LIN {X 0,Y 467.875,Z 296.784,A -85,B 0,C 180,E1 -7639.396,E2 -7639.396} C_VEL
LIN {X 0,Y 467.446,Z 305.686,A -85,B 0,C 180,E1 -7640.699,E2 -7640.699} C_VEL
LIN {X 0,Y 467.093,Z 312.847,A -85,B 0,C 180,E1 -7642,E2 -7642} C_VEL
LIN {X 0,Y 466.87,Z 319.224,A -85,B 0,C 180,E1 -7643.479,E2 -7643.479} C_VEL
LIN {X 0,Y 466.784,Z 323.676,A -85,B 0,C 180,E1 -7644.817,E2 -7644.817} C_VEL
LIN {X 0,Y 466.663,Z 325.957,A -85,B 0,C 180,E1 -7645.681,E2 -7645.681} C_VEL
LIN {X 0,Y 466.695,Z 327.806,A -85,B 0,C 180,E1 -7646.546,E2 -7646.546} C_VEL
LIN {X 0,Y 466.646,Z 329.192,A -85,B 0,C 180,E1 -7647.41,E2 -7647.41} C_VEL
LIN {X 0,Y 466.589,Z 330.785,A -85,B 0,C 180,E1 -7649.137,E2 -7649.137} C_VEL
LIN {X 0,Y 466.57,Z 331,A -85,B 0,C 180,E1 -7650,E2 -7650} C_VEL
LIN {X 0,Y 466.589,Z 330.786,A -85,B 0,C 180,E1 -7650.863,E2 -7650.863} C_VEL
LIN {X 0,Y 466.646,Z 329.196,A -85,B 0,C 180,E1 -7652.589,E2 -7652.589} C_VEL
LIN {X 0,Y 466.695,Z 327.81,A -85,B 0,C 180,E1 -7653.453,E2 -7653.453} C_VEL
LIN {X 0,Y 466.703,Z 324.896,A -85,B 0,C 180,E1 -7654.751,E2 -7654.751} C_VEL
LIN {X 0,Y 466.84,Z 320.949,A -85,B 0,C 180,E1 -7656.049,E2 -7656.049} C_VEL
LIN {X 0,Y 466.998,Z 314.876,A -85,B 0,C 180,E1 -7657.567,E2 -7657.567} C_VEL
LIN {X 0,Y 467.35,Z 308.236,A -85,B 0,C 180,E1 -7658.867,E2 -7658.867} C_VEL
LIN {X 0,Y 467.737,Z 299.994,A -85,B 0,C 180,E1 -7660.169,E2 -7660.169} C_VEL
LIN {X 0,Y 468.123,Z 291.523,A -85,B 0,C 180,E1 -7661.254,E2 -7661.254} C_VEL
LIN {X 0,Y 468.66,Z 281.242,A -85,B 0,C 180,E1 -7662.319,E2 -7662.319} C_VEL
LIN {X 0,Y 469.099,Z 269.657,A -85,B 0,C 180,E1 -7663.284,E2 -7663.284} C_VEL
LIN {X 0,Y 469.623,Z 257.36,A -85,B 0,C 180,E1 -7664.074,E2 -7664.074} C_VEL
LIN {X 0,Y 470.109,Z 245.016,A -85,B 0,C 180,E1 -7664.667,E2 -7664.667} C_VEL
LIN {X 0,Y 469.597,Z 238.804,A -85,B 0,C 180,E1 -7664.922,E2 -7664.922} C_VEL
LIN {X 0,Y 467.324,Z 225.956,A -85,B 0,C 180,E1 -7665.358,E2 -7665.358} C_VEL
LIN {X 0,Y 467.08,Z 224.269,A -85,B 0,C 180,E1 -7665.42,E2 -7665.42} C_VEL
LIN {X 0,Y 467.234,Z 216.192,A -85,B 0,C 180,E1 -7668.625,E2 -7668.625} C_VEL
LIN {X 0,Y 467.417,Z 208.755,A -85,B 0,C 180,E1 -7671.615,E2 -7671.615} C_VEL
LIN {X 0,Y 467.625,Z 201.974,A -85,B 0,C 180,E1 -7674.412,E2 -7674.412} C_VEL
LIN {X 0,Y 467.942,Z 194.095,A -85,B 0,C 180,E1 -7677.748,E2 -7677.748} C_VEL
LIN {X 0,Y 468.191,Z 187.326,A -85,B 0,C 180,E1 -7680.688,E2 -7680.688} C_VEL
LIN {X 0,Y 468.489,Z 180.565,A -85,B 0,C 180,E1 -7683.714,E2 -7683.714} C_VEL
LIN {X 0,Y 468.556,Z 175.849,A -85,B 0,C 180,E1 -7685.908,E2 -7685.908} C_VEL
LIN {X 0,Y 467.806,Z 170.377,A -85,B 0,C 180,E1 -7688.628,E2 -7688.628} C_VEL
LIN {X 0,Y 467.581,Z 169.245,A -85,B 0,C 180,E1 -7689.283,E2 -7689.283} C_VEL
LIN {X 0,Y 467.586,Z 169.242,A -85,B 0,C 180,E1 -7692.567,E2 -7692.567} C_VEL
LIN {X 0,Y 467.565,Z 169.245,A -85,B 0,C 180,E1 -7695.052,E2 -7695.052} C_VEL
LIN {X 0,Y 467.588,Z 169.24,A -85,B 0,C 180,E1 -7697.44,E2 -7697.44} C_VEL
LIN {X 0,Y 467.549,Z 169.245,A -85,B 0,C 180,E1 -7700.852,E2 -7700.852} C_VEL
LIN {X 0,Y 467.55,Z 169.247,A -85,B 0,C 180,E1 -7704.262,E2 -7704.262} C_VEL
LIN {X 0,Y 467.579,Z 169.241,A -85,B 0,C 180,E1 -7707.321,E2 -7707.321} C_VEL
LIN {X 0,Y 467.569,Z 169.244,A -85,B 0,C 180,E1 -7710.667,E2 -7710.667} C_VEL
LIN {X 0,Y 467.611,Z 169.237,A -85,B 0,C 180,E1 -7713.199,E2 -7713.199} C_VEL
LIN {X 0,Y 467.588,Z 169.238,A -85,B 0,C 180,E1 -7716.469,E2 -7716.469} C_VEL
LIN {X 0,Y 467.62,Z 169.237,A -85,B 0,C 180,E1 -7719.777,E2 -7719.777} C_VEL
LIN {X 0,Y 467.605,Z 169.238,A -85,B 0,C 180,E1 -7722.507,E2 -7722.507} C_VEL
LIN {X 0,Y 467.604,Z 169.239,A -85,B 0,C 180,E1 -7725.196,E2 -7725.196} C_VEL
LIN {X 0,Y 467.653,Z 169.234,A -85,B 0,C 180,E1 -7727.854,E2 -7727.854} C_VEL
LIN {X 0,Y 467.654,Z 169.235,A -85,B 0,C 180,E1 -7731.357,E2 -7731.357} C_VEL
LIN {X 0,Y 467.708,Z 169.223,A -85,B 0,C 180,E1 -7733.962,E2 -7733.962} C_VEL
LIN {X 0,Y 467.856,Z 169.206,A -85,B 0,C 180,E1 -7737.417,E2 -7737.417} C_VEL
LIN {X 0,Y 467.881,Z 169.204,A -85,B 0,C 180,E1 -7740,E2 -7740} C_VEL
LIN {X 0,Y 467.855,Z 169.207,A -85,B 0,C 180,E1 -7742.583,E2 -7742.583} C_VEL
LIN {X 0,Y 467.707,Z 169.224,A -85,B 0,C 180,E1 -7746.038,E2 -7746.038} C_VEL
LIN {X 0,Y 467.654,Z 169.234,A -85,B 0,C 180,E1 -7748.643,E2 -7748.643} C_VEL
LIN {X 0,Y 467.654,Z 169.236,A -85,B 0,C 180,E1 -7752.146,E2 -7752.146} C_VEL
LIN {X 0,Y 467.637,Z 169.236,A -85,B 0,C 180,E1 -7755.695,E2 -7755.695} C_VEL
LIN {X 0,Y 467.615,Z 169.237,A -85,B 0,C 180,E1 -7758.765,E2 -7758.765} C_VEL
LIN {X 0,Y 467.578,Z 169.241,A -85,B 0,C 180,E1 -7761.268,E2 -7761.268} C_VEL
LIN {X 0,Y 467.561,Z 169.247,A -85,B 0,C 180,E1 -7763.944,E2 -7763.944} C_VEL
LIN {X 0,Y 467.611,Z 169.235,A -85,B 0,C 180,E1 -7766.801,E2 -7766.801} C_VEL
LIN {X 0,Y 467.553,Z 169.245,A -85,B 0,C 180,E1 -7769.738,E2 -7769.738} C_VEL
LIN {X 0,Y 467.58,Z 169.242,A -85,B 0,C 180,E1 -7772.759,E2 -7772.759} C_VEL
LIN {X 0,Y 467.543,Z 169.247,A -85,B 0,C 180,E1 -7775.891,E2 -7775.891} C_VEL
LIN {X 0,Y 467.55,Z 169.247,A -85,B 0,C 180,E1 -7779.148,E2 -7779.148} C_VEL
LIN {X 0,Y 467.588,Z 169.24,A -85,B 0,C 180,E1 -7782.56,E2 -7782.56} C_VEL
LIN {X 0,Y 467.57,Z 169.243,A -85,B 0,C 180,E1 -7785.054,E2 -7785.054} C_VEL
LIN {X 0,Y 467.589,Z 169.241,A -85,B 0,C 180,E1 -7787.44,E2 -7787.44} C_VEL
LIN {X 0,Y 467.556,Z 169.245,A -85,B 0,C 180,E1 -7790.853,E2 -7790.853} C_VEL
LIN {X 0,Y 467.512,Z 169.254,A -85,B 0,C 180,E1 -7793.037,E2 -7793.037} C_VEL
LIN {X 0,Y 467.45,Z 169.259,A -85,B 0,C 180,E1 -7794.28,E2 -7794.28} C_VEL
LIN {X 0,Y 467.423,Z 171.585,A -85,B 0,C 180,E1 -7796.199,E2 -7796.199} C_VEL
LIN {X 0,Y 467.378,Z 175.811,A -85,B 0,C 180,E1 -7799.253,E2 -7799.253} C_VEL
LIN {X 0,Y 467.229,Z 180.015,A -85,B 0,C 180,E1 -7802.206,E2 -7802.206} C_VEL
LIN {X 0,Y 467.14,Z 184.191,A -85,B 0,C 180,E1 -7805.087,E2 -7805.087} C_VEL
LIN {X 0,Y 467.047,Z 188.346,A -85,B 0,C 180,E1 -7807.902,E2 -7807.902} C_VEL
LIN {X 0,Y 466.911,Z 192.566,A -85,B 0,C 180,E1 -7810.662,E2 -7810.662} C_VEL
LIN {X 0,Y 466.814,Z 197.398,A -85,B 0,C 180,E1 -7813.714,E2 -7813.714} C_VEL
LIN {X 0,Y 466.697,Z 198.811,A -85,B 0,C 180,E1 -7814.092,E2 -7814.092} C_VEL
LIN {X 0,Y 466.299,Z 202.019,A -85,B 0,C 180,E1 -7814.468,E2 -7814.468} C_VEL
LIN {X 0,Y 465.498,Z 207.579,A -85,B 0,C 180,E1 -7814.817,E2 -7814.817} C_VEL
LIN {X 0,Y 463.951,Z 218.12,A -85,B 0,C 180,E1 -7815.189,E2 -7815.189} C_VEL
LIN {X 0,Y 463.13,Z 225.353,A -85,B 0,C 180,E1 -7815.502,E2 -7815.502} C_VEL
LIN {X 0,Y 462.607,Z 236.688,A -85,B 0,C 180,E1 -7816.157,E2 -7816.157} C_VEL
LIN {X 0,Y 462.159,Z 248.349,A -85,B 0,C 180,E1 -7817.038,E2 -7817.038} C_VEL
LIN {X 0,Y 461.634,Z 258.814,A -85,B 0,C 180,E1 -7818.029,E2 -7818.029} C_VEL
LIN {X 0,Y 461.194,Z 267.362,A -85,B 0,C 180,E1 -7819.019,E2 -7819.019} C_VEL
LIN {X 0,Y 460.79,Z 275.235,A -85,B 0,C 180,E1 -7820.12,E2 -7820.12} C_VEL
LIN {X 0,Y 460.344,Z 282.934,A -85,B 0,C 180,E1 -7821.44,E2 -7821.44} C_VEL
LIN {X 0,Y 460.007,Z 289.993,A -85,B 0,C 180,E1 -7822.98,E2 -7822.98} C_VEL
LIN {X 0,Y 459.888,Z 294.695,A -85,B 0,C 180,E1 -7824.299,E2 -7824.299} C_VEL
LIN {X 0,Y 459.69,Z 298.298,A -85,B 0,C 180,E1 -7825.616,E2 -7825.616} C_VEL
LIN {X 0,Y 459.727,Z 300.157,A -85,B 0,C 180,E1 -7826.494,E2 -7826.494} C_VEL
LIN {X 0,Y 459.617,Z 301.562,A -85,B 0,C 180,E1 -7827.371,E2 -7827.371} C_VEL
LIN {X 0,Y 459.525,Z 303.175,A -85,B 0,C 180,E1 -7829.124,E2 -7829.124} C_VEL
LIN {X 0,Y 459.532,Z 303.41,A -85,B 0,C 180,E1 -7830,E2 -7830} C_VEL
LIN {X 0,Y 459.524,Z 303.224,A -85,B 0,C 180,E1 -7830.877,E2 -7830.877} C_VEL
LIN {X 0,Y 459.617,Z 301.675,A -85,B 0,C 180,E1 -7832.629,E2 -7832.629} C_VEL
LIN {X 0,Y 459.726,Z 300.319,A -85,B 0,C 180,E1 -7833.506,E2 -7833.506} C_VEL
LIN {X 0,Y 459.678,Z 297.461,A -85,B 0,C 180,E1 -7834.824,E2 -7834.824} C_VEL
LIN {X 0,Y 459.946,Z 293.575,A -85,B 0,C 180,E1 -7836.14,E2 -7836.14} C_VEL
LIN {X 0,Y 460.053,Z 288.569,A -85,B 0,C 180,E1 -7837.461,E2 -7837.461} C_VEL
LIN {X 0,Y 460.392,Z 282.263,A -85,B 0,C 180,E1 -7838.781,E2 -7838.781} C_VEL
LIN {X 0,Y 460.813,Z 274.368,A -85,B 0,C 180,E1 -7840.102,E2 -7840.102} C_VEL
LIN {X 0,Y 461.215,Z 266.319,A -85,B 0,C 180,E1 -7841.203,E2 -7841.203} C_VEL
LIN {X 0,Y 461.777,Z 256.494,A -85,B 0,C 180,E1 -7842.303,E2 -7842.303} C_VEL
LIN {X 0,Y 462.242,Z 245.72,A -85,B 0,C 180,E1 -7843.274,E2 -7843.274} C_VEL
LIN {X 0,Y 462.781,Z 234.616,A -85,B 0,C 180,E1 -7844.063,E2 -7844.063} C_VEL
LIN {X 0,Y 463.246,Z 222.652,A -85,B 0,C 180,E1 -7844.721,E2 -7844.721} C_VEL
LIN {X 0,Y 463.261,Z 216.269,A -85,B 0,C 180,E1 -7845.008,E2 -7845.008} C_VEL
LIN {X 0,Y 460.768,Z 203.666,A -85,B 0,C 180,E1 -7845.517,E2 -7845.517} C_VEL
LIN {X 0,Y 459.757,Z 199.146,A -85,B 0,C 180,E1 -7845.666,E2 -7845.666} C_VEL
LIN {X 0,Y 459.844,Z 194.325,A -85,B 0,C 180,E1 -7848.721,E2 -7848.721} C_VEL
LIN {X 0,Y 459.918,Z 190.074,A -85,B 0,C 180,E1 -7851.515,E2 -7851.515} C_VEL
LIN {X 0,Y 460.07,Z 185.88,A -85,B 0,C 180,E1 -7854.359,E2 -7854.359} C_VEL
LIN {X 0,Y 460.171,Z 181.159,A -85,B 0,C 180,E1 -7857.648,E2 -7857.648} C_VEL
LIN {X 0,Y 460.291,Z 177.484,A -85,B 0,C 180,E1 -7860.256,E2 -7860.256} C_VEL
LIN {X 0,Y 460.372,Z 173.244,A -85,B 0,C 180,E1 -7863.338,E2 -7863.338} C_VEL
LIN {X 0,Y 460.43,Z 170.397,A -85,B 0,C 180,E1 -7865.453,E2 -7865.453} C_VEL
LIN {X 0,Y 460.48,Z 170.127,A -85,B 0,C 180,E1 -7867.473,E2 -7867.473} C_VEL
LIN {X 0,Y 460.525,Z 170.12,A -85,B 0,C 180,E1 -7870.266,E2 -7870.266} C_VEL
LIN {X 0,Y 460.505,Z 170.124,A -85,B 0,C 180,E1 -7873.375,E2 -7873.375} C_VEL
LIN {X 0,Y 460.5,Z 170.122,A -85,B 0,C 180,E1 -7876.624,E2 -7876.624} C_VEL
LIN {X 0,Y 460.539,Z 170.116,A -85,B 0,C 180,E1 -7879.731,E2 -7879.731} C_VEL
LIN {X 0,Y 460.482,Z 170.128,A -85,B 0,C 180,E1 -7882.527,E2 -7882.527} C_VEL
LIN {X 0,Y 460.535,Z 170.119,A -85,B 0,C 180,E1 -7885.623,E2 -7885.623} C_VEL
LIN {X 0,Y 460.539,Z 170.12,A -85,B 0,C 180,E1 -7888.744,E2 -7888.744} C_VEL
LIN {X 0,Y 460.583,Z 170.114,A -85,B 0,C 180,E1 -7892.254,E2 -7892.254} C_VEL
LIN {X 0,Y 460.541,Z 170.117,A -85,B 0,C 180,E1 -7894.704,E2 -7894.704} C_VEL
LIN {X 0,Y 460.511,Z 170.121,A -85,B 0,C 180,E1 -7897.571,E2 -7897.571} C_VEL
LIN {X 0,Y 460.569,Z 170.115,A -85,B 0,C 180,E1 -7900.384,E2 -7900.384} C_VEL
LIN {X 0,Y 460.601,Z 170.111,A -85,B 0,C 180,E1 -7904.002,E2 -7904.002} C_VEL
LIN {X 0,Y 460.61,Z 170.111,A -85,B 0,C 180,E1 -7907.666,E2 -7907.666} C_VEL
LIN {X 0,Y 460.61,Z 170.109,A -85,B 0,C 180,E1 -7911.223,E2 -7911.223} C_VEL
LIN {X 0,Y 460.674,Z 170.101,A -85,B 0,C 180,E1 -7913.87,E2 -7913.87} C_VEL
LIN {X 0,Y 460.797,Z 170.087,A -85,B 0,C 180,E1 -7917.377,E2 -7917.377} C_VEL
LIN {X 0,Y 460.855,Z 170.079,A -85,B 0,C 180,E1 -7920,E2 -7920} C_VEL
LIN {X 0,Y 460.799,Z 170.086,A -85,B 0,C 180,E1 -7922.622,E2 -7922.622} C_VEL
LIN {X 0,Y 460.676,Z 170.099,A -85,B 0,C 180,E1 -7926.13,E2 -7926.13} C_VEL
LIN {X 0,Y 460.609,Z 170.113,A -85,B 0,C 180,E1 -7928.777,E2 -7928.777} C_VEL
LIN {X 0,Y 460.636,Z 170.108,A -85,B 0,C 180,E1 -7932.457,E2 -7932.457} C_VEL
LIN {X 0,Y 460.601,Z 170.112,A -85,B 0,C 180,E1 -7935.998,E2 -7935.998} C_VEL
LIN {X 0,Y 460.569,Z 170.114,A -85,B 0,C 180,E1 -7939.616,E2 -7939.616} C_VEL
LIN {X 0,Y 460.511,Z 170.123,A -85,B 0,C 180,E1 -7942.429,E2 -7942.429} C_VEL
LIN {X 0,Y 460.553,Z 170.119,A -85,B 0,C 180,E1 -7945.798,E2 -7945.798} C_VEL
LIN {X 0,Y 460.553,Z 170.117,A -85,B 0,C 180,E1 -7948.233,E2 -7948.233} C_VEL
LIN {X 0,Y 460.522,Z 170.122,A -85,B 0,C 180,E1 -7951.283,E2 -7951.283} C_VEL
LIN {X 0,Y 460.53,Z 170.119,A -85,B 0,C 180,E1 -7954.505,E2 -7954.505} C_VEL
LIN {X 0,Y 460.483,Z 170.129,A -85,B 0,C 180,E1 -7957.625,E2 -7957.625} C_VEL
LIN {X 0,Y 460.531,Z 170.12,A -85,B 0,C 180,E1 -7961.011,E2 -7961.011} C_VEL
LIN {X 0,Y 460.508,Z 170.124,A -85,B 0,C 180,E1 -7964.169,E2 -7964.169} C_VEL
LIN {X 0,Y 460.514,Z 170.12,A -85,B 0,C 180,E1 -7967.1,E2 -7967.1} C_VEL
LIN {X 0,Y 460.542,Z 170.122,A -85,B 0,C 180,E1 -7970.392,E2 -7970.392} C_VEL
LIN {X 0,Y 460.585,Z 170.311,A -85,B 0,C 180,E1 -7970.649,E2 -7970.649} C_VEL
LIN {X 0,Y 461.488,Z 176.003,A -85,B 0,C 180,E1 -7973.563,E2 -7973.563} C_VEL
LIN {X 0,Y 461.531,Z 180.472,A -85,B 0,C 180,E1 -7975.707,E2 -7975.707} C_VEL
LIN {X 0,Y 461.234,Z 187.215,A -85,B 0,C 180,E1 -7978.797,E2 -7978.797} C_VEL
LIN {X 0,Y 460.951,Z 193.981,A -85,B 0,C 180,E1 -7981.794,E2 -7981.794} C_VEL
LIN {X 0,Y 460.653,Z 200.735,A -85,B 0,C 180,E1 -7984.711,E2 -7984.711} C_VEL
LIN {X 0,Y 460.422,Z 207.527,A -85,B 0,C 180,E1 -7987.567,E2 -7987.567} C_VEL
LIN {X 0,Y 460.202,Z 215.596,A -85,B 0,C 180,E1 -7990.878,E2 -7990.878} C_VEL
LIN {X 0,Y 460.029,Z 224.29,A -85,B 0,C 180,E1 -7994.364,E2 -7994.364} C_VEL
LIN {X 0,Y 462.399,Z 237.666,A -85,B 0,C 180,E1 -7994.806,E2 -7994.806} C_VEL
LIN {X 0,Y 463.229,Z 244.803,A -85,B 0,C 180,E1 -7995.109,E2 -7995.109} C_VEL
LIN {X 0,Y 462.786,Z 257.144,A -85,B 0,C 180,E1 -7995.713,E2 -7995.713} C_VEL
LIN {X 0,Y 462.22,Z 269.005,A -85,B 0,C 180,E1 -7996.48,E2 -7996.48} C_VEL
LIN {X 0,Y 461.765,Z 279.345,A -85,B 0,C 180,E1 -7997.334,E2 -7997.334} C_VEL
LIN {X 0,Y 461.267,Z 289.356,A -85,B 0,C 180,E1 -7998.353,E2 -7998.353} C_VEL
LIN {X 0,Y 460.754,Z 298.208,A -85,B 0,C 180,E1 -7999.453,E2 -7999.453} C_VEL
LIN {X 0,Y 460.346,Z 306.844,A -85,B 0,C 180,E1 -8000.775,E2 -8000.775} C_VEL
LIN {X 0,Y 459.98,Z 313.745,A -85,B 0,C 180,E1 -8002.096,E2 -8002.096} C_VEL
LIN {X 0,Y 459.8,Z 319.492,A -85,B 0,C 180,E1 -8003.475,E2 -8003.475} C_VEL
LIN {X 0,Y 459.701,Z 323.619,A -85,B 0,C 180,E1 -8004.737,E2 -8004.737} C_VEL
LIN {X 0,Y 459.58,Z 325.915,A -85,B 0,C 180,E1 -8005.615,E2 -8005.615} C_VEL
LIN {X 0,Y 459.591,Z 327.779,A -85,B 0,C 180,E1 -8006.493,E2 -8006.493} C_VEL
LIN {X 0,Y 459.57,Z 329.176,A -85,B 0,C 180,E1 -8007.37,E2 -8007.37} C_VEL
LIN {X 0,Y 459.494,Z 330.779,A -85,B 0,C 180,E1 -8009.123,E2 -8009.123} C_VEL
LIN {X 0,Y 459.474,Z 330.994,A -85,B 0,C 180,E1 -8010,E2 -8010} C_VEL
LIN {X 0,Y 459.494,Z 330.779,A -85,B 0,C 180,E1 -8010.876,E2 -8010.876} C_VEL
LIN {X 0,Y 459.57,Z 329.179,A -85,B 0,C 180,E1 -8012.629,E2 -8012.629} C_VEL
LIN {X 0,Y 459.591,Z 327.783,A -85,B 0,C 180,E1 -8013.507,E2 -8013.507} C_VEL
LIN {X 0,Y 459.634,Z 324.846,A -85,B 0,C 180,E1 -8014.824,E2 -8014.824} C_VEL
LIN {X 0,Y 459.758,Z 320.873,A -85,B 0,C 180,E1 -8016.142,E2 -8016.142} C_VEL
LIN {X 0,Y 459.929,Z 314.76,A -85,B 0,C 180,E1 -8017.684,E2 -8017.684} C_VEL
LIN {X 0,Y 460.305,Z 308.084,A -85,B 0,C 180,E1 -8019.003,E2 -8019.003} C_VEL
LIN {X 0,Y 460.698,Z 299.799,A -85,B 0,C 180,E1 -8020.326,E2 -8020.326} C_VEL
LIN {X 0,Y 461.133,Z 291.309,A -85,B 0,C 180,E1 -8021.427,E2 -8021.427} C_VEL
LIN {X 0,Y 461.678,Z 281.197,A -85,B 0,C 180,E1 -8022.493,E2 -8022.493} C_VEL
LIN {X 0,Y 462.116,Z 270.731,A -85,B 0,C 180,E1 -8023.388,E2 -8023.388} C_VEL
LIN {X 0,Y 462.631,Z 259.068,A -85,B 0,C 180,E1 -8024.179,E2 -8024.179} C_VEL
LIN {X 0,Y 463.133,Z 247.407,A -85,B 0,C 180,E1 -8024.781,E2 -8024.781} C_VEL
LIN {X 0,Y 463.006,Z 241.858,A -85,B 0,C 180,E1 -8025.02,E2 -8025.02} C_VEL
LIN {X 0,Y 460.834,Z 229.016,A -85,B 0,C 180,E1 -8025.501,E2 -8025.501} C_VEL
LIN {X 0,Y 460.019,Z 224.117,A -85,B 0,C 180,E1 -8025.662,E2 -8025.662} C_VEL
LIN {X 0,Y 460.2,Z 215.549,A -85,B 0,C 180,E1 -8029.121,E2 -8029.121} C_VEL
LIN {X 0,Y 460.42,Z 207.462,A -85,B 0,C 180,E1 -8032.433,E2 -8032.433} C_VEL
LIN {X 0,Y 460.738,Z 199.434,A -85,B 0,C 180,E1 -8035.845,E2 -8035.845} C_VEL
LIN {X 0,Y 460.986,Z 192.849,A -85,B 0,C 180,E1 -8038.7,E2 -8038.7} C_VEL
LIN {X 0,Y 461.258,Z 186.702,A -85,B 0,C 180,E1 -8041.433,E2 -8041.433} C_VEL
LIN {X 0,Y 461.584,Z 179.604,A -85,B 0,C 180,E1 -8044.695,E2 -8044.695} C_VEL
LIN {X 0,Y 461.493,Z 175.986,A -85,B 0,C 180,E1 -8046.436,E2 -8046.436} C_VEL
LIN {X 0,Y 460.549,Z 170.122,A -85,B 0,C 180,E1 -8049.481,E2 -8049.481} C_VEL
LIN {X 0,Y 460.522,Z 170.123,A -85,B 0,C 180,E1 -8052.181,E2 -8052.181} C_VEL
LIN {X 0,Y 460.512,Z 170.122,A -85,B 0,C 180,E1 -8055.411,E2 -8055.411} C_VEL
LIN {X 0,Y 460.531,Z 170.12,A -85,B 0,C 180,E1 -8058.397,E2 -8058.397} C_VEL
LIN {X 0,Y 460.503,Z 170.12,A -85,B 0,C 180,E1 -8061.264,E2 -8061.264} C_VEL
LIN {X 0,Y 460.502,Z 170.123,A -85,B 0,C 180,E1 -8064.554,E2 -8064.554} C_VEL
LIN {X 0,Y 460.529,Z 170.121,A -85,B 0,C 180,E1 -8067.715,E2 -8067.715} C_VEL
LIN {X 0,Y 460.538,Z 170.119,A -85,B 0,C 180,E1 -8070.769,E2 -8070.769} C_VEL
LIN {X 0,Y 460.554,Z 170.117,A -85,B 0,C 180,E1 -8073.734,E2 -8073.734} C_VEL
LIN {X 0,Y 460.542,Z 170.115,A -85,B 0,C 180,E1 -8076.624,E2 -8076.624} C_VEL
LIN {X 0,Y 460.549,Z 170.119,A -85,B 0,C 180,E1 -8079.453,E2 -8079.453} C_VEL
LIN {X 0,Y 460.556,Z 170.117,A -85,B 0,C 180,E1 -8082.23,E2 -8082.23} C_VEL
LIN {X 0,Y 460.563,Z 170.117,A -85,B 0,C 180,E1 -8084.965,E2 -8084.965} C_VEL
LIN {X 0,Y 460.606,Z 170.11,A -85,B 0,C 180,E1 -8088.559,E2 -8088.559} C_VEL
LIN {X 0,Y 460.606,Z 170.112,A -85,B 0,C 180,E1 -8091.223,E2 -8091.223} C_VEL
LIN {X 0,Y 460.672,Z 170.099,A -85,B 0,C 180,E1 -8093.87,E2 -8093.87} C_VEL
LIN {X 0,Y 460.796,Z 170.086,A -85,B 0,C 180,E1 -8097.378,E2 -8097.378} C_VEL
LIN {X 0,Y 460.852,Z 170.079,A -85,B 0,C 180,E1 -8100,E2 -8100} C_VEL
LIN {X 0,Y 460.796,Z 170.087,A -85,B 0,C 180,E1 -8102.623,E2 -8102.623} C_VEL
LIN {X 0,Y 460.672,Z 170.101,A -85,B 0,C 180,E1 -8106.13,E2 -8106.13} C_VEL
LIN {X 0,Y 460.606,Z 170.11,A -85,B 0,C 180,E1 -8108.777,E2 -8108.777} C_VEL
LIN {X 0,Y 460.611,Z 170.11,A -85,B 0,C 180,E1 -8112.445,E2 -8112.445} C_VEL
LIN {X 0,Y 460.598,Z 170.112,A -85,B 0,C 180,E1 -8115.998,E2 -8115.998} C_VEL
LIN {X 0,Y 460.569,Z 170.114,A -85,B 0,C 180,E1 -8118.902,E2 -8118.902} C_VEL
LIN {X 0,Y 460.514,Z 170.121,A -85,B 0,C 180,E1 -8121.486,E2 -8121.486} C_VEL
LIN {X 0,Y 460.529,Z 170.118,A -85,B 0,C 180,E1 -8124.333,E2 -8124.333} C_VEL
LIN {X 0,Y 460.587,Z 170.114,A -85,B 0,C 180,E1 -8127.748,E2 -8127.748} C_VEL
LIN {X 0,Y 460.519,Z 170.123,A -85,B 0,C 180,E1 -8131.283,E2 -8131.283} C_VEL
LIN {X 0,Y 460.527,Z 170.12,A -85,B 0,C 180,E1 -8134.505,E2 -8134.505} C_VEL
LIN {X 0,Y 460.482,Z 170.127,A -85,B 0,C 180,E1 -8137.625,E2 -8137.625} C_VEL
LIN {X 0,Y 460.537,Z 170.116,A -85,B 0,C 180,E1 -8140.269,E2 -8140.269} C_VEL
LIN {X 0,Y 460.497,Z 170.123,A -85,B 0,C 180,E1 -8143.376,E2 -8143.376} C_VEL
LIN {X 0,Y 460.5,Z 170.125,A -85,B 0,C 180,E1 -8146.625,E2 -8146.625} C_VEL
LIN {X 0,Y 460.538,Z 170.118,A -85,B 0,C 180,E1 -8149.732,E2 -8149.732} C_VEL
LIN {X 0,Y 460.491,Z 170.125,A -85,B 0,C 180,E1 -8152.526,E2 -8152.526} C_VEL
LIN {X 0,Y 460.371,Z 170.266,A -85,B 0,C 180,E1 -8154.542,E2 -8154.542} C_VEL
LIN {X 0,Y 460.345,Z 173.703,A -85,B 0,C 180,E1 -8157.106,E2 -8157.106} C_VEL
LIN {X 0,Y 460.29,Z 177.344,A -85,B 0,C 180,E1 -8159.744,E2 -8159.744} C_VEL
LIN {X 0,Y 460.169,Z 181.546,A -85,B 0,C 180,E1 -8162.731,E2 -8162.731} C_VEL
LIN {X 0,Y 460.071,Z 185.729,A -85,B 0,C 180,E1 -8165.642,E2 -8165.642} C_VEL
LIN {X 0,Y 459.963,Z 190.324,A -85,B 0,C 180,E1 -8168.757,E2 -8168.757} C_VEL
LIN {X 0,Y 459.794,Z 195.597,A -85,B 0,C 180,E1 -8172.2,E2 -8172.2} C_VEL
LIN {X 0,Y 459.79,Z 199.144,A -85,B 0,C 180,E1 -8174.427,E2 -8174.427} C_VEL
LIN {X 0,Y 462.626,Z 212.526,A -85,B 0,C 180,E1 -8174.921,E2 -8174.921} C_VEL
LIN {X 0,Y 463.362,Z 218.158,A -85,B 0,C 180,E1 -8175.17,E2 -8175.17} C_VEL
LIN {X 0,Y 463.13,Z 225.353,A -85,B 0,C 180,E1 -8175.502,E2 -8175.502} C_VEL
LIN {X 0,Y 462.255,Z 230.79,A -85,B 0,C 180,E1 -8175.768,E2 -8175.768} C_VEL
LIN {X 0,Y 459.168,Z 239.456,A -85,B 0,C 180,E1 -8176.227,E2 -8176.227} C_VEL
LIN {X 0,Y 456.036,Z 247.721,A -85,B 0,C 180,E1 -8176.781,E2 -8176.781} C_VEL
LIN {X 0,Y 455.097,Z 252.526,A -85,B 0,C 180,E1 -8177.194,E2 -8177.194} C_VEL
LIN {X 0,Y 454.553,Z 262.05,A -85,B 0,C 180,E1 -8178.179,E2 -8178.179} C_VEL
LIN {X 0,Y 454.07,Z 270.894,A -85,B 0,C 180,E1 -8179.296,E2 -8179.296} C_VEL
LIN {X 0,Y 453.584,Z 279.522,A -85,B 0,C 180,E1 -8180.637,E2 -8180.637} C_VEL
LIN {X 0,Y 453.133,Z 286.4,A -85,B 0,C 180,E1 -8181.976,E2 -8181.976} C_VEL
LIN {X 0,Y 452.899,Z 291.798,A -85,B 0,C 180,E1 -8183.287,E2 -8183.287} C_VEL
LIN {X 0,Y 452.702,Z 296.226,A -85,B 0,C 180,E1 -8184.656,E2 -8184.656} C_VEL
LIN {X 0,Y 452.599,Z 298.513,A -85,B 0,C 180,E1 -8185.547,E2 -8185.547} C_VEL
LIN {X 0,Y 452.641,Z 300.371,A -85,B 0,C 180,E1 -8186.439,E2 -8186.439} C_VEL
LIN {X 0,Y 452.544,Z 301.775,A -85,B 0,C 180,E1 -8187.33,E2 -8187.33} C_VEL
LIN {X 0,Y 452.432,Z 303.389,A -85,B 0,C 180,E1 -8189.11,E2 -8189.11} C_VEL
LIN {X 0,Y 452.437,Z 303.623,A -85,B 0,C 180,E1 -8190,E2 -8190} C_VEL
LIN {X 0,Y 452.432,Z 303.437,A -85,B 0,C 180,E1 -8190.89,E2 -8190.89} C_VEL
LIN {X 0,Y 452.544,Z 301.887,A -85,B 0,C 180,E1 -8192.671,E2 -8192.671} C_VEL
LIN {X 0,Y 452.64,Z 300.531,A -85,B 0,C 180,E1 -8193.561,E2 -8193.561} C_VEL
LIN {X 0,Y 452.609,Z 297.672,A -85,B 0,C 180,E1 -8194.899,E2 -8194.899} C_VEL
LIN {X 0,Y 452.874,Z 293.787,A -85,B 0,C 180,E1 -8196.237,E2 -8196.237} C_VEL
LIN {X 0,Y 452.998,Z 288.781,A -85,B 0,C 180,E1 -8197.578,E2 -8197.578} C_VEL
LIN {X 0,Y 453.381,Z 282.474,A -85,B 0,C 180,E1 -8198.918,E2 -8198.918} C_VEL
LIN {X 0,Y 453.807,Z 274.578,A -85,B 0,C 180,E1 -8200.259,E2 -8200.259} C_VEL
LIN {X 0,Y 454.253,Z 266.529,A -85,B 0,C 180,E1 -8201.377,E2 -8201.377} C_VEL
LIN {X 0,Y 454.831,Z 256.703,A -85,B 0,C 180,E1 -8202.494,E2 -8202.494} C_VEL
LIN {X 0,Y 455.391,Z 245.359,A -85,B 0,C 180,E1 -8203.523,E2 -8203.523} C_VEL
LIN {X 0,Y 455.901,Z 234.822,A -85,B 0,C 180,E1 -8204.28,E2 -8204.28} C_VEL
LIN {X 0,Y 456.399,Z 222.855,A -85,B 0,C 180,E1 -8204.947,E2 -8204.947} C_VEL
LIN {X 0,Y 456.282,Z 216.534,A -85,B 0,C 180,E1 -8205.24,E2 -8205.24} C_VEL
LIN {X 0,Y 453.764,Z 204.067,A -85,B 0,C 180,E1 -8205.757,E2 -8205.757} C_VEL
LIN {X 0,Y 452.697,Z 199.349,A -85,B 0,C 180,E1 -8205.918,E2 -8205.918} C_VEL
LIN {X 0,Y 452.782,Z 194.512,A -85,B 0,C 180,E1 -8209.024,E2 -8209.024} C_VEL
LIN {X 0,Y 452.884,Z 190.245,A -85,B 0,C 180,E1 -8211.866,E2 -8211.866} C_VEL
LIN {X 0,Y 453.008,Z 186.038,A -85,B 0,C 180,E1 -8214.764,E2 -8214.764} C_VEL
LIN {X 0,Y 453.119,Z 181.66,A -85,B 0,C 180,E1 -8217.86,E2 -8217.86} C_VEL
LIN {X 0,Y 453.26,Z 177.606,A -85,B 0,C 180,E1 -8220.776,E2 -8220.776} C_VEL
LIN {X 0,Y 453.355,Z 173.347,A -85,B 0,C 180,E1 -8223.923,E2 -8223.923} C_VEL
LIN {X 0,Y 453.386,Z 171.926,A -85,B 0,C 180,E1 -8224.998,E2 -8224.998} C_VEL
LIN {X 0,Y 453.405,Z 171.009,A -85,B 0,C 180,E1 -8226.29,E2 -8226.29} C_VEL
LIN {X 0,Y 453.442,Z 171.003,A -85,B 0,C 180,E1 -8229.455,E2 -8229.455} C_VEL
LIN {X 0,Y 453.45,Z 171.002,A -85,B 0,C 180,E1 -8231.931,E2 -8231.931} C_VEL
LIN {X 0,Y 453.486,Z 170.998,A -85,B 0,C 180,E1 -8235.471,E2 -8235.471} C_VEL
LIN {X 0,Y 453.481,Z 170.995,A -85,B 0,C 180,E1 -8238.209,E2 -8238.209} C_VEL
LIN {X 0,Y 453.465,Z 171.003,A -85,B 0,C 180,E1 -8240.798,E2 -8240.798} C_VEL
LIN {X 0,Y 453.444,Z 171.001,A -85,B 0,C 180,E1 -8243.916,E2 -8243.916} C_VEL
LIN {X 0,Y 453.479,Z 170.999,A -85,B 0,C 180,E1 -8247.151,E2 -8247.151} C_VEL
LIN {X 0,Y 453.476,Z 170.998,A -85,B 0,C 180,E1 -8250.268,E2 -8250.268} C_VEL
LIN {X 0,Y 453.503,Z 170.993,A -85,B 0,C 180,E1 -8253.294,E2 -8253.294} C_VEL
LIN {X 0,Y 453.499,Z 170.998,A -85,B 0,C 180,E1 -8256.238,E2 -8256.238} C_VEL
LIN {X 0,Y 453.483,Z 170.996,A -85,B 0,C 180,E1 -8259.118,E2 -8259.118} C_VEL
LIN {X 0,Y 453.505,Z 170.995,A -85,B 0,C 180,E1 -8261.944,E2 -8261.944} C_VEL
LIN {X 0,Y 453.541,Z 170.99,A -85,B 0,C 180,E1 -8264.726,E2 -8264.726} C_VEL
LIN {X 0,Y 453.559,Z 170.987,A -85,B 0,C 180,E1 -8268.379,E2 -8268.379} C_VEL
LIN {X 0,Y 453.577,Z 170.984,A -85,B 0,C 180,E1 -8271.086,E2 -8271.086} C_VEL
LIN {X 0,Y 453.64,Z 170.977,A -85,B 0,C 180,E1 -8273.774,E2 -8273.774} C_VEL
LIN {X 0,Y 453.741,Z 170.966,A -85,B 0,C 180,E1 -8277.337,E2 -8277.337} C_VEL
LIN {X 0,Y 453.825,Z 170.954,A -85,B 0,C 180,E1 -8280,E2 -8280} C_VEL
LIN {X 0,Y 453.743,Z 170.965,A -85,B 0,C 180,E1 -8282.663,E2 -8282.663} C_VEL
LIN {X 0,Y 453.642,Z 170.975,A -85,B 0,C 180,E1 -8286.226,E2 -8286.226} C_VEL
LIN {X 0,Y 453.577,Z 170.987,A -85,B 0,C 180,E1 -8288.914,E2 -8288.914} C_VEL
LIN {X 0,Y 453.603,Z 170.984,A -85,B 0,C 180,E1 -8292.551,E2 -8292.551} C_VEL
LIN {X 0,Y 453.545,Z 170.99,A -85,B 0,C 180,E1 -8296.196,E2 -8296.196} C_VEL
LIN {X 0,Y 453.518,Z 170.992,A -85,B 0,C 180,E1 -8299.039,E2 -8299.039} C_VEL
LIN {X 0,Y 453.477,Z 170.997,A -85,B 0,C 180,E1 -8301.836,E2 -8301.836} C_VEL
LIN {X 0,Y 453.501,Z 170.994,A -85,B 0,C 180,E1 -8304.735,E2 -8304.735} C_VEL
LIN {X 0,Y 453.533,Z 170.992,A -85,B 0,C 180,E1 -8307.96,E2 -8307.96} C_VEL
LIN {X 0,Y 453.467,Z 171,A -85,B 0,C 180,E1 -8311.525,E2 -8311.525} C_VEL
LIN {X 0,Y 453.486,Z 170.996,A -85,B 0,C 180,E1 -8314.777,E2 -8314.777} C_VEL
LIN {X 0,Y 453.446,Z 170.999,A -85,B 0,C 180,E1 -8318.314,E2 -8318.314} C_VEL
LIN {X 0,Y 453.495,Z 170.994,A -85,B 0,C 180,E1 -8320.609,E2 -8320.609} C_VEL
LIN {X 0,Y 453.455,Z 171.003,A -85,B 0,C 180,E1 -8323.244,E2 -8323.244} C_VEL
LIN {X 0,Y 453.465,Z 171.001,A -85,B 0,C 180,E1 -8325.779,E2 -8325.779} C_VEL
LIN {X 0,Y 453.481,Z 170.999,A -85,B 0,C 180,E1 -8328.209,E2 -8328.209} C_VEL
LIN {X 0,Y 453.549,Z 171.185,A -85,B 0,C 180,E1 -8330.412,E2 -8330.412} C_VEL
LIN {X 0,Y 454.484,Z 177.158,A -85,B 0,C 180,E1 -8333.525,E2 -8333.525} C_VEL
LIN {X 0,Y 454.535,Z 181.493,A -85,B 0,C 180,E1 -8335.642,E2 -8335.642} C_VEL
LIN {X 0,Y 454.226,Z 188.287,A -85,B 0,C 180,E1 -8338.806,E2 -8338.806} C_VEL
LIN {X 0,Y 453.892,Z 195.295,A -85,B 0,C 180,E1 -8341.955,E2 -8341.955} C_VEL
LIN {X 0,Y 453.558,Z 202.871,A -85,B 0,C 180,E1 -8345.268,E2 -8345.268} C_VEL
LIN {X 0,Y 453.286,Z 210.437,A -85,B 0,C 180,E1 -8348.478,E2 -8348.478} C_VEL
LIN {X 0,Y 453.123,Z 216.741,A -85,B 0,C 180,E1 -8351.106,E2 -8351.106} C_VEL
LIN {X 0,Y 452.932,Z 223.96,A -85,B 0,C 180,E1 -8354.107,E2 -8354.107} C_VEL
LIN {X 0,Y 455.336,Z 237.519,A -85,B 0,C 180,E1 -8354.567,E2 -8354.567} C_VEL
LIN {X 0,Y 456.345,Z 245.893,A -85,B 0,C 180,E1 -8354.937,E2 -8354.937} C_VEL
LIN {X 0,Y 455.886,Z 256.93,A -85,B 0,C 180,E1 -8355.492,E2 -8355.492} C_VEL
LIN {X 0,Y 455.303,Z 268.791,A -85,B 0,C 180,E1 -8356.271,E2 -8356.271} C_VEL
LIN {X 0,Y 454.776,Z 279.444,A -85,B 0,C 180,E1 -8357.167,E2 -8357.167} C_VEL
LIN {X 0,Y 454.293,Z 289.142,A -85,B 0,C 180,E1 -8358.171,E2 -8358.171} C_VEL
LIN {X 0,Y 453.735,Z 297.994,A -85,B 0,C 180,E1 -8359.288,E2 -8359.288} C_VEL
LIN {X 0,Y 453.31,Z 306.63,A -85,B 0,C 180,E1 -8360.631,E2 -8360.631} C_VEL
LIN {X 0,Y 452.924,Z 313.531,A -85,B 0,C 180,E1 -8361.972,E2 -8361.972} C_VEL
LIN {X 0,Y 452.71,Z 319.714,A -85,B 0,C 180,E1 -8363.493,E2 -8363.493} C_VEL
LIN {X 0,Y 452.567,Z 324.631,A -85,B 0,C 180,E1 -8365.1,E2 -8365.1} C_VEL
LIN {X 0,Y 452.488,Z 327.565,A -85,B 0,C 180,E1 -8366.438,E2 -8366.438} C_VEL
LIN {X 0,Y 452.496,Z 328.963,A -85,B 0,C 180,E1 -8367.329,E2 -8367.329} C_VEL
LIN {X 0,Y 452.403,Z 330.566,A -85,B 0,C 180,E1 -8369.11,E2 -8369.11} C_VEL
LIN {X 0,Y 452.381,Z 330.783,A -85,B 0,C 180,E1 -8370,E2 -8370} C_VEL
LIN {X 0,Y 452.403,Z 330.567,A -85,B 0,C 180,E1 -8370.89,E2 -8370.89} C_VEL
LIN {X 0,Y 452.496,Z 328.967,A -85,B 0,C 180,E1 -8372.67,E2 -8372.67} C_VEL
LIN {X 0,Y 452.488,Z 327.57,A -85,B 0,C 180,E1 -8373.562,E2 -8373.562} C_VEL
LIN {X 0,Y 452.567,Z 324.634,A -85,B 0,C 180,E1 -8374.899,E2 -8374.899} C_VEL
LIN {X 0,Y 452.687,Z 319.805,A -85,B 0,C 180,E1 -8376.482,E2 -8376.482} C_VEL
LIN {X 0,Y 452.926,Z 313.534,A -85,B 0,C 180,E1 -8378.027,E2 -8378.027} C_VEL
LIN {X 0,Y 453.31,Z 306.632,A -85,B 0,C 180,E1 -8379.369,E2 -8379.369} C_VEL
LIN {X 0,Y 453.733,Z 297.997,A -85,B 0,C 180,E1 -8380.712,E2 -8380.712} C_VEL
LIN {X 0,Y 454.281,Z 289.145,A -85,B 0,C 180,E1 -8381.828,E2 -8381.828} C_VEL
LIN {X 0,Y 454.836,Z 279.311,A -85,B 0,C 180,E1 -8382.845,E2 -8382.845} C_VEL
LIN {X 0,Y 455.258,Z 268.798,A -85,B 0,C 180,E1 -8383.73,E2 -8383.73} C_VEL
LIN {X 0,Y 455.843,Z 256.933,A -85,B 0,C 180,E1 -8384.509,E2 -8384.509} C_VEL
LIN {X 0,Y 456.341,Z 244.589,A -85,B 0,C 180,E1 -8385.12,E2 -8385.12} C_VEL
LIN {X 0,Y 454.285,Z 231.745,A -85,B 0,C 180,E1 -8385.653,E2 -8385.653} C_VEL
LIN {X 0,Y 452.934,Z 223.957,A -85,B 0,C 180,E1 -8385.894,E2 -8385.894} C_VEL
LIN {X 0,Y 453.155,Z 215.286,A -85,B 0,C 180,E1 -8389.478,E2 -8389.478} C_VEL
LIN {X 0,Y 453.405,Z 207.344,A -85,B 0,C 180,E1 -8392.799,E2 -8392.799} C_VEL
LIN {X 0,Y 453.687,Z 199.854,A -85,B 0,C 180,E1 -8396.042,E2 -8396.042} C_VEL
LIN {X 0,Y 453.999,Z 192.726,A -85,B 0,C 180,E1 -8399.184,E2 -8399.184} C_VEL
LIN {X 0,Y 454.325,Z 185.977,A -85,B 0,C 180,E1 -8402.254,E2 -8402.254} C_VEL
LIN {X 0,Y 454.621,Z 179.248,A -85,B 0,C 180,E1 -8405.429,E2 -8405.429} C_VEL
LIN {X 0,Y 454.315,Z 175.9,A -85,B 0,C 180,E1 -8407.107,E2 -8407.107} C_VEL
LIN {X 0,Y 453.512,Z 170.998,A -85,B 0,C 180,E1 -8409.735,E2 -8409.735} C_VEL
LIN {X 0,Y 453.462,Z 171.001,A -85,B 0,C 180,E1 -8412.995,E2 -8412.995} C_VEL
LIN {X 0,Y 453.461,Z 170.999,A -85,B 0,C 180,E1 -8415.778,E2 -8415.778} C_VEL
LIN {X 0,Y 453.478,Z 170.997,A -85,B 0,C 180,E1 -8418.209,E2 -8418.209} C_VEL
LIN {X 0,Y 453.462,Z 171,A -85,B 0,C 180,E1 -8420.798,E2 -8420.798} C_VEL
LIN {X 0,Y 453.442,Z 171.003,A -85,B 0,C 180,E1 -8423.916,E2 -8423.916} C_VEL
LIN {X 0,Y 453.487,Z 170.997,A -85,B 0,C 180,E1 -8426.811,E2 -8426.811} C_VEL
LIN {X 0,Y 453.473,Z 171,A -85,B 0,C 180,E1 -8430.268,E2 -8430.268} C_VEL
LIN {X 0,Y 453.5,Z 170.995,A -85,B 0,C 180,E1 -8433.293,E2 -8433.293} C_VEL
LIN {X 0,Y 453.495,Z 170.995,A -85,B 0,C 180,E1 -8436.238,E2 -8436.238} C_VEL
LIN {X 0,Y 453.48,Z 170.996,A -85,B 0,C 180,E1 -8439.117,E2 -8439.117} C_VEL
LIN {X 0,Y 453.508,Z 170.994,A -85,B 0,C 180,E1 -8441.944,E2 -8441.944} C_VEL
LIN {X 0,Y 453.538,Z 170.99,A -85,B 0,C 180,E1 -8444.726,E2 -8444.726} C_VEL
LIN {X 0,Y 453.556,Z 170.987,A -85,B 0,C 180,E1 -8448.379,E2 -8448.379} C_VEL
LIN {X 0,Y 453.574,Z 170.987,A -85,B 0,C 180,E1 -8451.086,E2 -8451.086} C_VEL
LIN {X 0,Y 453.639,Z 170.976,A -85,B 0,C 180,E1 -8453.774,E2 -8453.774} C_VEL
LIN {X 0,Y 453.74,Z 170.965,A -85,B 0,C 180,E1 -8457.337,E2 -8457.337} C_VEL
LIN {X 0,Y 453.822,Z 170.955,A -85,B 0,C 180,E1 -8460,E2 -8460} C_VEL
LIN {X 0,Y 453.74,Z 170.966,A -85,B 0,C 180,E1 -8462.663,E2 -8462.663} C_VEL
LIN {X 0,Y 453.639,Z 170.977,A -85,B 0,C 180,E1 -8466.226,E2 -8466.226} C_VEL
LIN {X 0,Y 453.574,Z 170.985,A -85,B 0,C 180,E1 -8468.914,E2 -8468.914} C_VEL
LIN {X 0,Y 453.561,Z 170.988,A -85,B 0,C 180,E1 -8472.529,E2 -8472.529} C_VEL
LIN {X 0,Y 453.543,Z 170.99,A -85,B 0,C 180,E1 -8476.196,E2 -8476.196} C_VEL
LIN {X 0,Y 453.518,Z 170.992,A -85,B 0,C 180,E1 -8479.041,E2 -8479.041} C_VEL
LIN {X 0,Y 453.474,Z 170.999,A -85,B 0,C 180,E1 -8481.836,E2 -8481.836} C_VEL
LIN {X 0,Y 453.499,Z 170.992,A -85,B 0,C 180,E1 -8484.735,E2 -8484.735} C_VEL
LIN {X 0,Y 453.536,Z 170.991,A -85,B 0,C 180,E1 -8487.961,E2 -8487.961} C_VEL
LIN {X 0,Y 453.464,Z 171,A -85,B 0,C 180,E1 -8491.525,E2 -8491.525} C_VEL
LIN {X 0,Y 453.483,Z 170.998,A -85,B 0,C 180,E1 -8494.777,E2 -8494.777} C_VEL
LIN {X 0,Y 453.446,Z 171,A -85,B 0,C 180,E1 -8498.314,E2 -8498.314} C_VEL
LIN {X 0,Y 453.493,Z 170.994,A -85,B 0,C 180,E1 -8500.609,E2 -8500.609} C_VEL
LIN {X 0,Y 453.454,Z 171.001,A -85,B 0,C 180,E1 -8503.244,E2 -8503.244} C_VEL
LIN {X 0,Y 453.466,Z 170.999,A -85,B 0,C 180,E1 -8505.779,E2 -8505.779} C_VEL
LIN {X 0,Y 453.479,Z 170.998,A -85,B 0,C 180,E1 -8508.21,E2 -8508.21} C_VEL
LIN {X 0,Y 453.469,Z 171,A -85,B 0,C 180,E1 -8510.798,E2 -8510.798} C_VEL
LIN {X 0,Y 453.385,Z 171.011,A -85,B 0,C 180,E1 -8513.911,E2 -8513.911} C_VEL
LIN {X 0,Y 453.362,Z 172.12,A -85,B 0,C 180,E1 -8515.246,E2 -8515.246} C_VEL
LIN {X 0,Y 453.271,Z 176.5,A -85,B 0,C 180,E1 -8518.516,E2 -8518.516} C_VEL
LIN {X 0,Y 453.177,Z 180.289,A -85,B 0,C 180,E1 -8521.266,E2 -8521.266} C_VEL
LIN {X 0,Y 453.033,Z 184.496,A -85,B 0,C 180,E1 -8524.255,E2 -8524.255} C_VEL
LIN {X 0,Y 452.935,Z 188.68,A -85,B 0,C 180,E1 -8527.176,E2 -8527.176} C_VEL
LIN {X 0,Y 452.8,Z 192.928,A -85,B 0,C 180,E1 -8530.034,E2 -8530.034} C_VEL
LIN {X 0,Y 452.7,Z 197.252,A -85,B 0,C 180,E1 -8532.845,E2 -8532.845} C_VEL
LIN {X 0,Y 452.743,Z 199.496,A -85,B 0,C 180,E1 -8534.184,E2 -8534.184} C_VEL
LIN {X 0,Y 455.619,Z 212.763,A -85,B 0,C 180,E1 -8534.684,E2 -8534.684} C_VEL
LIN {X 0,Y 456.509,Z 218.382,A -85,B 0,C 180,E1 -8534.943,E2 -8534.943} C_VEL
LIN {X 0,Y 456.087,Z 229.629,A -85,B 0,C 180,E1 -8535.499,E2 -8535.499} C_VEL
LIN {X 0,Y 455.581,Z 241.137,A -85,B 0,C 180,E1 -8536.243,E2 -8536.243} C_VEL
LIN {X 0,Y 455.175,Z 251.363,A -85,B 0,C 180,E1 -8537.084,E2 -8537.084} C_VEL
LIN {X 0,Y 455.097,Z 252.526,A -85,B 0,C 180,E1 -8537.194,E2 -8537.194} C_VEL
LIN {X 0,Y 454.123,Z 257.281,A -85,B 0,C 180,E1 -8537.637,E2 -8537.637} C_VEL
LIN {X 0,Y 450.829,Z 264.667,A -85,B 0,C 180,E1 -8538.376,E2 -8538.376} C_VEL
LIN {X 0,Y 447.641,Z 271.455,A -85,B 0,C 180,E1 -8539.191,E2 -8539.191} C_VEL
LIN {X 0,Y 446.824,Z 275.273,A -85,B 0,C 180,E1 -8539.747,E2 -8539.747} C_VEL
LIN {X 0,Y 446.388,Z 282.191,A -85,B 0,C 180,E1 -8540.942,E2 -8540.942} C_VEL
LIN {X 0,Y 446.001,Z 288.614,A -85,B 0,C 180,E1 -8542.303,E2 -8542.303} C_VEL
LIN {X 0,Y 445.828,Z 293.706,A -85,B 0,C 180,E1 -8543.665,E2 -8543.665} C_VEL
LIN {X 0,Y 445.553,Z 297.666,A -85,B 0,C 180,E1 -8545.023,E2 -8545.023} C_VEL
LIN {X 0,Y 445.557,Z 300.585,A -85,B 0,C 180,E1 -8546.383,E2 -8546.383} C_VEL
LIN {X 0,Y 445.473,Z 301.988,A -85,B 0,C 180,E1 -8547.287,E2 -8547.287} C_VEL
LIN {X 0,Y 445.342,Z 303.602,A -85,B 0,C 180,E1 -8549.096,E2 -8549.096} C_VEL
LIN {X 0,Y 445.344,Z 303.836,A -85,B 0,C 180,E1 -8550,E2 -8550} C_VEL
LIN {X 0,Y 445.342,Z 303.65,A -85,B 0,C 180,E1 -8550.904,E2 -8550.904} C_VEL
LIN {X 0,Y 445.473,Z 302.099,A -85,B 0,C 180,E1 -8552.713,E2 -8552.713} C_VEL
LIN {X 0,Y 445.556,Z 300.743,A -85,B 0,C 180,E1 -8553.618,E2 -8553.618} C_VEL
LIN {X 0,Y 445.546,Z 297.884,A -85,B 0,C 180,E1 -8554.977,E2 -8554.977} C_VEL
LIN {X 0,Y 445.808,Z 293.999,A -85,B 0,C 180,E1 -8556.336,E2 -8556.336} C_VEL
LIN {X 0,Y 445.967,Z 288.992,A -85,B 0,C 180,E1 -8557.698,E2 -8557.698} C_VEL
LIN {X 0,Y 446.372,Z 282.684,A -85,B 0,C 180,E1 -8559.059,E2 -8559.059} C_VEL
LIN {X 0,Y 446.821,Z 274.788,A -85,B 0,C 180,E1 -8560.421,E2 -8560.421} C_VEL
LIN {X 0,Y 447.422,Z 264.964,A -85,B 0,C 180,E1 -8561.783,E2 -8561.783} C_VEL
LIN {X 0,Y 448.026,Z 254.983,A -85,B 0,C 180,E1 -8562.884,E2 -8562.884} C_VEL
LIN {X 0,Y 448.584,Z 243.575,A -85,B 0,C 180,E1 -8563.894,E2 -8563.894} C_VEL
LIN {X 0,Y 449.112,Z 233.267,A -85,B 0,C 180,E1 -8564.616,E2 -8564.616} C_VEL
LIN {X 0,Y 449.591,Z 221.931,A -85,B 0,C 180,E1 -8565.237,E2 -8565.237} C_VEL
LIN {X 0,Y 449.514,Z 218.103,A -85,B 0,C 180,E1 -8565.414,E2 -8565.414} C_VEL
LIN {X 0,Y 446.866,Z 204.961,A -85,B 0,C 180,E1 -8565.989,E2 -8565.989} C_VEL
LIN {X 0,Y 445.603,Z 199.528,A -85,B 0,C 180,E1 -8566.196,E2 -8566.196} C_VEL
LIN {X 0,Y 445.717,Z 194.7,A -85,B 0,C 180,E1 -8569.337,E2 -8569.337} C_VEL
LIN {X 0,Y 445.819,Z 190.419,A -85,B 0,C 180,E1 -8572.231,E2 -8572.231} C_VEL
LIN {X 0,Y 445.94,Z 186.196,A -85,B 0,C 180,E1 -8575.184,E2 -8575.184} C_VEL
LIN {X 0,Y 446.087,Z 181.988,A -85,B 0,C 180,E1 -8578.206,E2 -8578.206} C_VEL
LIN {X 0,Y 446.215,Z 177.731,A -85,B 0,C 180,E1 -8581.316,E2 -8581.316} C_VEL
LIN {X 0,Y 446.328,Z 173.453,A -85,B 0,C 180,E1 -8584.532,E2 -8584.532} C_VEL
LIN {X 0,Y 446.319,Z 172.026,A -85,B 0,C 180,E1 -8585.635,E2 -8585.635} C_VEL
LIN {X 0,Y 446.398,Z 171.88,A -85,B 0,C 180,E1 -8588.076,E2 -8588.076} C_VEL
LIN {X 0,Y 446.408,Z 171.88,A -85,B 0,C 180,E1 -8591.393,E2 -8591.393} C_VEL
LIN {X 0,Y 446.453,Z 171.874,A -85,B 0,C 180,E1 -8595.104,E2 -8595.104} C_VEL
LIN {X 0,Y 446.43,Z 171.876,A -85,B 0,C 180,E1 -8598.609,E2 -8598.609} C_VEL
LIN {X 0,Y 446.4,Z 171.878,A -85,B 0,C 180,E1 -8601.923,E2 -8601.923} C_VEL
LIN {X 0,Y 446.421,Z 171.876,A -85,B 0,C 180,E1 -8605.476,E2 -8605.476} C_VEL
LIN {X 0,Y 446.417,Z 171.879,A -85,B 0,C 180,E1 -8608.7,E2 -8608.7} C_VEL
LIN {X 0,Y 446.486,Z 171.868,A -85,B 0,C 180,E1 -8611.821,E2 -8611.821} C_VEL
LIN {X 0,Y 446.445,Z 171.872,A -85,B 0,C 180,E1 -8614.847,E2 -8614.847} C_VEL
LIN {X 0,Y 446.449,Z 171.874,A -85,B 0,C 180,E1 -8618.245,E2 -8618.245} C_VEL
LIN {X 0,Y 446.453,Z 171.875,A -85,B 0,C 180,E1 -8621.649,E2 -8621.649} C_VEL
LIN {X 0,Y 446.509,Z 171.866,A -85,B 0,C 180,E1 -8624.48,E2 -8624.48} C_VEL
LIN {X 0,Y 446.518,Z 171.865,A -85,B 0,C 180,E1 -8628.193,E2 -8628.193} C_VEL
LIN {X 0,Y 446.526,Z 171.862,A -85,B 0,C 180,E1 -8630.944,E2 -8630.944} C_VEL
LIN {X 0,Y 446.609,Z 171.854,A -85,B 0,C 180,E1 -8633.676,E2 -8633.676} C_VEL
LIN {X 0,Y 446.688,Z 171.845,A -85,B 0,C 180,E1 -8637.295,E2 -8637.295} C_VEL
LIN {X 0,Y 446.795,Z 171.83,A -85,B 0,C 180,E1 -8640,E2 -8640} C_VEL
LIN {X 0,Y 446.69,Z 171.843,A -85,B 0,C 180,E1 -8642.705,E2 -8642.705} C_VEL
LIN {X 0,Y 446.611,Z 171.851,A -85,B 0,C 180,E1 -8646.324,E2 -8646.324} C_VEL
LIN {X 0,Y 446.526,Z 171.864,A -85,B 0,C 180,E1 -8649.056,E2 -8649.056} C_VEL
LIN {X 0,Y 446.535,Z 171.863,A -85,B 0,C 180,E1 -8652.729,E2 -8652.729} C_VEL
LIN {X 0,Y 446.49,Z 171.869,A -85,B 0,C 180,E1 -8656.459,E2 -8656.459} C_VEL
LIN {X 0,Y 446.469,Z 171.869,A -85,B 0,C 180,E1 -8659.303,E2 -8659.303} C_VEL
LIN {X 0,Y 446.419,Z 171.88,A -85,B 0,C 180,E1 -8662.2,E2 -8662.2} C_VEL
LIN {X 0,Y 446.444,Z 171.872,A -85,B 0,C 180,E1 -8665.153,E2 -8665.153} C_VEL
LIN {X 0,Y 446.486,Z 171.869,A -85,B 0,C 180,E1 -8668.179,E2 -8668.179} C_VEL
LIN {X 0,Y 446.42,Z 171.878,A -85,B 0,C 180,E1 -8671.775,E2 -8671.775} C_VEL
LIN {X 0,Y 446.427,Z 171.875,A -85,B 0,C 180,E1 -8674.523,E2 -8674.523} C_VEL
LIN {X 0,Y 446.398,Z 171.878,A -85,B 0,C 180,E1 -8678.076,E2 -8678.076} C_VEL
LIN {X 0,Y 446.429,Z 171.878,A -85,B 0,C 180,E1 -8681.391,E2 -8681.391} C_VEL
LIN {X 0,Y 446.453,Z 171.875,A -85,B 0,C 180,E1 -8685.104,E2 -8685.104} C_VEL
LIN {X 0,Y 446.43,Z 171.877,A -85,B 0,C 180,E1 -8688.609,E2 -8688.609} C_VEL
LIN {X 0,Y 446.495,Z 172.064,A -85,B 0,C 180,E1 -8690.172,E2 -8690.172} C_VEL
LIN {X 0,Y 447.439,Z 178.038,A -85,B 0,C 180,E1 -8693.354,E2 -8693.354} C_VEL
LIN {X 0,Y 447.624,Z 180.779,A -85,B 0,C 180,E1 -8694.73,E2 -8694.73} C_VEL
LIN {X 0,Y 447.276,Z 187.711,A -85,B 0,C 180,E1 -8698.049,E2 -8698.049} C_VEL
LIN {X 0,Y 446.982,Z 193.733,A -85,B 0,C 180,E1 -8700.829,E2 -8700.829} C_VEL
LIN {X 0,Y 446.659,Z 200.499,A -85,B 0,C 180,E1 -8703.86,E2 -8703.86} C_VEL
LIN {X 0,Y 446.33,Z 208.391,A -85,B 0,C 180,E1 -8707.308,E2 -8707.308} C_VEL
LIN {X 0,Y 446.083,Z 216.263,A -85,B 0,C 180,E1 -8710.679,E2 -8710.679} C_VEL
LIN {X 0,Y 445.873,Z 223.732,A -85,B 0,C 180,E1 -8713.845,E2 -8713.845} C_VEL
LIN {X 0,Y 448.324,Z 237.615,A -85,B 0,C 180,E1 -8714.331,E2 -8714.331} C_VEL
LIN {X 0,Y 449.447,Z 246.983,A -85,B 0,C 180,E1 -8714.758,E2 -8714.758} C_VEL
LIN {X 0,Y 448.905,Z 258.638,A -85,B 0,C 180,E1 -8715.377,E2 -8715.377} C_VEL
LIN {X 0,Y 448.29,Z 270.007,A -85,B 0,C 180,E1 -8716.168,E2 -8716.168} C_VEL
LIN {X 0,Y 447.737,Z 281.207,A -85,B 0,C 180,E1 -8717.155,E2 -8717.155} C_VEL
LIN {X 0,Y 447.179,Z 290.878,A -85,B 0,C 180,E1 -8718.211,E2 -8718.211} C_VEL
LIN {X 0,Y 446.642,Z 299.367,A -85,B 0,C 180,E1 -8719.345,E2 -8719.345} C_VEL
LIN {X 0,Y 446.193,Z 307.653,A -85,B 0,C 180,E1 -8720.709,E2 -8720.709} C_VEL
LIN {X 0,Y 445.806,Z 314.33,A -85,B 0,C 180,E1 -8722.071,E2 -8722.071} C_VEL
LIN {X 0,Y 445.598,Z 320.445,A -85,B 0,C 180,E1 -8723.661,E2 -8723.661} C_VEL
LIN {X 0,Y 445.5,Z 324.419,A -85,B 0,C 180,E1 -8725.022,E2 -8725.022} C_VEL
LIN {X 0,Y 445.387,Z 327.352,A -85,B 0,C 180,E1 -8726.381,E2 -8726.381} C_VEL
LIN {X 0,Y 445.422,Z 328.75,A -85,B 0,C 180,E1 -8727.287,E2 -8727.287} C_VEL
LIN {X 0,Y 445.315,Z 330.354,A -85,B 0,C 180,E1 -8729.095,E2 -8729.095} C_VEL
LIN {X 0,Y 445.292,Z 330.57,A -85,B 0,C 180,E1 -8730,E2 -8730} C_VEL
LIN {X 0,Y 445.315,Z 330.354,A -85,B 0,C 180,E1 -8730.904,E2 -8730.904} C_VEL
LIN {X 0,Y 445.422,Z 328.754,A -85,B 0,C 180,E1 -8732.713,E2 -8732.713} C_VEL
LIN {X 0,Y 445.387,Z 327.356,A -85,B 0,C 180,E1 -8733.619,E2 -8733.619} C_VEL
LIN {X 0,Y 445.5,Z 324.421,A -85,B 0,C 180,E1 -8734.977,E2 -8734.977} C_VEL
LIN {X 0,Y 445.585,Z 320.079,A -85,B 0,C 180,E1 -8736.449,E2 -8736.449} C_VEL
LIN {X 0,Y 445.807,Z 314.332,A -85,B 0,C 180,E1 -8737.928,E2 -8737.928} C_VEL
LIN {X 0,Y 446.193,Z 307.655,A -85,B 0,C 180,E1 -8739.291,E2 -8739.291} C_VEL
LIN {X 0,Y 446.64,Z 299.37,A -85,B 0,C 180,E1 -8740.654,E2 -8740.654} C_VEL
LIN {X 0,Y 447.173,Z 290.882,A -85,B 0,C 180,E1 -8741.789,E2 -8741.789} C_VEL
LIN {X 0,Y 447.745,Z 281.144,A -85,B 0,C 180,E1 -8742.851,E2 -8742.851} C_VEL
LIN {X 0,Y 448.257,Z 270.014,A -85,B 0,C 180,E1 -8743.833,E2 -8743.833} C_VEL
LIN {X 0,Y 448.866,Z 258.642,A -85,B 0,C 180,E1 -8744.624,E2 -8744.624} C_VEL
LIN {X 0,Y 449.391,Z 246.98,A -85,B 0,C 180,E1 -8745.244,E2 -8745.244} C_VEL
LIN {X 0,Y 448.777,Z 240.417,A -85,B 0,C 180,E1 -8745.546,E2 -8745.546} C_VEL
LIN {X 0,Y 446.3,Z 226.481,A -85,B 0,C 180,E1 -8746.072,E2 -8746.072} C_VEL
LIN {X 0,Y 445.873,Z 223.731,A -85,B 0,C 180,E1 -8746.155,E2 -8746.155} C_VEL
LIN {X 0,Y 446.121,Z 215.137,A -85,B 0,C 180,E1 -8749.797,E2 -8749.797} C_VEL
LIN {X 0,Y 446.38,Z 207.253,A -85,B 0,C 180,E1 -8753.179,E2 -8753.179} C_VEL
LIN {X 0,Y 446.69,Z 199.349,A -85,B 0,C 180,E1 -8756.648,E2 -8756.648} C_VEL
LIN {X 0,Y 447.035,Z 192.633,A -85,B 0,C 180,E1 -8759.668,E2 -8759.668} C_VEL
LIN {X 0,Y 447.327,Z 186.985,A -85,B 0,C 180,E1 -8762.288,E2 -8762.288} C_VEL
LIN {X 0,Y 447.621,Z 180.265,A -85,B 0,C 180,E1 -8765.515,E2 -8765.515} C_VEL
LIN {X 0,Y 447.119,Z 175.805,A -85,B 0,C 180,E1 -8767.808,E2 -8767.808} C_VEL
LIN {X 0,Y 446.474,Z 171.875,A -85,B 0,C 180,E1 -8770.012,E2 -8770.012} C_VEL
LIN {X 0,Y 446.428,Z 171.877,A -85,B 0,C 180,E1 -8772.604,E2 -8772.604} C_VEL
LIN {X 0,Y 446.45,Z 171.876,A -85,B 0,C 180,E1 -8775.103,E2 -8775.103} C_VEL
LIN {X 0,Y 446.427,Z 171.879,A -85,B 0,C 180,E1 -8778.609,E2 -8778.609} C_VEL
LIN {X 0,Y 446.397,Z 171.878,A -85,B 0,C 180,E1 -8781.923,E2 -8781.923} C_VEL
LIN {X 0,Y 446.425,Z 171.875,A -85,B 0,C 180,E1 -8785.476,E2 -8785.476} C_VEL
LIN {X 0,Y 446.414,Z 171.879,A -85,B 0,C 180,E1 -8788.699,E2 -8788.699} C_VEL
LIN {X 0,Y 446.483,Z 171.87,A -85,B 0,C 180,E1 -8791.821,E2 -8791.821} C_VEL
LIN {X 0,Y 446.442,Z 171.872,A -85,B 0,C 180,E1 -8794.847,E2 -8794.847} C_VEL
LIN {X 0,Y 446.446,Z 171.873,A -85,B 0,C 180,E1 -8798.245,E2 -8798.245} C_VEL
LIN {X 0,Y 446.455,Z 171.874,A -85,B 0,C 180,E1 -8801.649,E2 -8801.649} C_VEL
LIN {X 0,Y 446.506,Z 171.866,A -85,B 0,C 180,E1 -8804.48,E2 -8804.48} C_VEL
LIN {X 0,Y 446.514,Z 171.864,A -85,B 0,C 180,E1 -8808.193,E2 -8808.193} C_VEL
LIN {X 0,Y 446.523,Z 171.864,A -85,B 0,C 180,E1 -8810.944,E2 -8810.944} C_VEL
LIN {X 0,Y 446.608,Z 171.852,A -85,B 0,C 180,E1 -8813.676,E2 -8813.676} C_VEL
LIN {X 0,Y 446.687,Z 171.844,A -85,B 0,C 180,E1 -8817.295,E2 -8817.295} C_VEL
LIN {X 0,Y 446.792,Z 171.83,A -85,B 0,C 180,E1 -8820,E2 -8820} C_VEL
LIN {X 0,Y 446.687,Z 171.845,A -85,B 0,C 180,E1 -8822.705,E2 -8822.705} C_VEL
LIN {X 0,Y 446.608,Z 171.854,A -85,B 0,C 180,E1 -8826.324,E2 -8826.324} C_VEL
LIN {X 0,Y 446.523,Z 171.862,A -85,B 0,C 180,E1 -8829.056,E2 -8829.056} C_VEL
LIN {X 0,Y 446.519,Z 171.864,A -85,B 0,C 180,E1 -8832.73,E2 -8832.73} C_VEL
LIN {X 0,Y 446.494,Z 171.869,A -85,B 0,C 180,E1 -8836.228,E2 -8836.228} C_VEL
LIN {X 0,Y 446.467,Z 171.871,A -85,B 0,C 180,E1 -8839.303,E2 -8839.303} C_VEL
LIN {X 0,Y 446.416,Z 171.879,A -85,B 0,C 180,E1 -8842.2,E2 -8842.2} C_VEL
LIN {X 0,Y 446.442,Z 171.872,A -85,B 0,C 180,E1 -8845.153,E2 -8845.153} C_VEL
LIN {X 0,Y 446.483,Z 171.869,A -85,B 0,C 180,E1 -8848.179,E2 -8848.179} C_VEL
LIN {X 0,Y 446.418,Z 171.878,A -85,B 0,C 180,E1 -8851.775,E2 -8851.775} C_VEL
LIN {X 0,Y 446.425,Z 171.876,A -85,B 0,C 180,E1 -8854.524,E2 -8854.524} C_VEL
LIN {X 0,Y 446.397,Z 171.878,A -85,B 0,C 180,E1 -8858.077,E2 -8858.077} C_VEL
LIN {X 0,Y 446.427,Z 171.876,A -85,B 0,C 180,E1 -8861.391,E2 -8861.391} C_VEL
LIN {X 0,Y 446.453,Z 171.874,A -85,B 0,C 180,E1 -8865.104,E2 -8865.104} C_VEL
LIN {X 0,Y 446.428,Z 171.877,A -85,B 0,C 180,E1 -8868.609,E2 -8868.609} C_VEL
LIN {X 0,Y 446.424,Z 171.879,A -85,B 0,C 180,E1 -8870.971,E2 -8870.971} C_VEL
LIN {X 0,Y 446.372,Z 171.886,A -85,B 0,C 180,E1 -8873.416,E2 -8873.416} C_VEL
LIN {X 0,Y 446.3,Z 171.905,A -85,B 0,C 180,E1 -8874.363,E2 -8874.363} C_VEL
LIN {X 0,Y 446.219,Z 176.174,A -85,B 0,C 180,E1 -8877.622,E2 -8877.622} C_VEL
LIN {X 0,Y 446.141,Z 180.428,A -85,B 0,C 180,E1 -8880.769,E2 -8880.769} C_VEL
LIN {X 0,Y 445.994,Z 184.795,A -85,B 0,C 180,E1 -8883.924,E2 -8883.924} C_VEL
LIN {X 0,Y 445.885,Z 188.849,A -85,B 0,C 180,E1 -8886.794,E2 -8886.794} C_VEL
LIN {X 0,Y 445.764,Z 193.111,A -85,B 0,C 180,E1 -8889.705,E2 -8889.705} C_VEL
LIN {X 0,Y 445.648,Z 197.448,A -85,B 0,C 180,E1 -8892.565,E2 -8892.565} C_VEL
LIN {X 0,Y 445.653,Z 199.769,A -85,B 0,C 180,E1 -8893.926,E2 -8893.926} C_VEL
LIN {X 0,Y 448.519,Z 212.651,A -85,B 0,C 180,E1 -8894.422,E2 -8894.422} C_VEL
LIN {X 0,Y 449.646,Z 219.902,A -85,B 0,C 180,E1 -8894.765,E2 -8894.765} C_VEL
LIN {X 0,Y 449.126,Z 231.828,A -85,B 0,C 180,E1 -8895.385,E2 -8895.385} C_VEL
LIN {X 0,Y 448.549,Z 243.592,A -85,B 0,C 180,E1 -8896.2,E2 -8896.2} C_VEL
LIN {X 0,Y 448.022,Z 254.999,A -85,B 0,C 180,E1 -8897.21,E2 -8897.21} C_VEL
LIN {X 0,Y 447.455,Z 264.211,A -85,B 0,C 180,E1 -8898.218,E2 -8898.218} C_VEL
LIN {X 0,Y 446.984,Z 272.71,A -85,B 0,C 180,E1 -8899.354,E2 -8899.354} C_VEL
LIN {X 0,Y 446.824,Z 275.273,A -85,B 0,C 180,E1 -8899.747,E2 -8899.747} C_VEL
LIN {X 0,Y 446.003,Z 278.949,A -85,B 0,C 180,E1 -8900.33,E2 -8900.33} C_VEL
LIN {X 0,Y 442.806,Z 284.489,A -85,B 0,C 180,E1 -8901.308,E2 -8901.308} C_VEL
LIN {X 0,Y 439.6,Z 289.447,A -85,B 0,C 180,E1 -8902.351,E2 -8902.351} C_VEL
LIN {X 0,Y 438.778,Z 292.081,A -85,B 0,C 180,E1 -8903.032,E2 -8903.032} C_VEL
LIN {X 0,Y 438.613,Z 296.654,A -85,B 0,C 180,E1 -8904.483,E2 -8904.483} C_VEL
LIN {X 0,Y 438.436,Z 298.942,A -85,B 0,C 180,E1 -8905.403,E2 -8905.403} C_VEL
LIN {X 0,Y 438.46,Z 300.799,A -85,B 0,C 180,E1 -8906.324,E2 -8906.324} C_VEL
LIN {X 0,Y 438.404,Z 302.201,A -85,B 0,C 180,E1 -8907.244,E2 -8907.244} C_VEL
LIN {X 0,Y 438.256,Z 303.815,A -85,B 0,C 180,E1 -8909.081,E2 -8909.081} C_VEL
LIN {X 0,Y 438.255,Z 304.049,A -85,B 0,C 180,E1 -8910,E2 -8910} C_VEL
LIN {X 0,Y 438.256,Z 303.862,A -85,B 0,C 180,E1 -8910.919,E2 -8910.919} C_VEL
LIN {X 0,Y 438.404,Z 302.31,A -85,B 0,C 180,E1 -8912.757,E2 -8912.757} C_VEL
LIN {X 0,Y 438.458,Z 300.956,A -85,B 0,C 180,E1 -8913.676,E2 -8913.676} C_VEL
LIN {X 0,Y 438.488,Z 298.096,A -85,B 0,C 180,E1 -8915.058,E2 -8915.058} C_VEL
LIN {X 0,Y 438.742,Z 294.211,A -85,B 0,C 180,E1 -8916.438,E2 -8916.438} C_VEL
LIN {X 0,Y 438.915,Z 289.203,A -85,B 0,C 180,E1 -8917.823,E2 -8917.823} C_VEL
LIN {X 0,Y 439.342,Z 282.895,A -85,B 0,C 180,E1 -8919.205,E2 -8919.205} C_VEL
LIN {X 0,Y 439.844,Z 274.998,A -85,B 0,C 180,E1 -8920.589,E2 -8920.589} C_VEL
LIN {X 0,Y 440.468,Z 265.173,A -85,B 0,C 180,E1 -8921.972,E2 -8921.972} C_VEL
LIN {X 0,Y 441.11,Z 255.304,A -85,B 0,C 180,E1 -8923.079,E2 -8923.079} C_VEL
LIN {X 0,Y 441.646,Z 244.656,A -85,B 0,C 180,E1 -8924.044,E2 -8924.044} C_VEL
LIN {X 0,Y 442.267,Z 233.472,A -85,B 0,C 180,E1 -8924.847,E2 -8924.847} C_VEL
LIN {X 0,Y 442.746,Z 222.135,A -85,B 0,C 180,E1 -8925.479,E2 -8925.479} C_VEL
LIN {X 0,Y 442.484,Z 218.311,A -85,B 0,C 180,E1 -8925.665,E2 -8925.665} C_VEL
LIN {X 0,Y 440.018,Z 206.086,A -85,B 0,C 180,E1 -8926.217,E2 -8926.217} C_VEL
LIN {X 0,Y 438.538,Z 199.745,A -85,B 0,C 180,E1 -8926.454,E2 -8926.454} C_VEL
LIN {X 0,Y 438.656,Z 194.888,A -85,B 0,C 180,E1 -8929.661,E2 -8929.661} C_VEL
LIN {X 0,Y 438.79,Z 190.592,A -85,B 0,C 180,E1 -8932.607,E2 -8932.607} C_VEL
LIN {X 0,Y 438.884,Z 186.354,A -85,B 0,C 180,E1 -8935.618,E2 -8935.618} C_VEL
LIN {X 0,Y 439.048,Z 182.135,A -85,B 0,C 180,E1 -8938.7,E2 -8938.7} C_VEL
LIN {X 0,Y 439.148,Z 179.294,A -85,B 0,C 180,E1 -8940.805,E2 -8940.805} C_VEL
LIN {X 0,Y 439.256,Z 174.997,A -85,B 0,C 180,E1 -8944.055,E2 -8944.055} C_VEL
LIN {X 0,Y 439.309,Z 173.367,A -85,B 0,C 180,E1 -8945.324,E2 -8945.324} C_VEL
LIN {X 0,Y 439.306,Z 172.766,A -85,B 0,C 180,E1 -8946.294,E2 -8946.294} C_VEL
LIN {X 0,Y 439.355,Z 172.756,A -85,B 0,C 180,E1 -8948.598,E2 -8948.598} C_VEL
LIN {X 0,Y 439.36,Z 172.756,A -85,B 0,C 180,E1 -8952.209,E2 -8952.209} C_VEL
LIN {X 0,Y 439.401,Z 172.754,A -85,B 0,C 180,E1 -8955.27,E2 -8955.27} C_VEL
LIN {X 0,Y 439.39,Z 172.754,A -85,B 0,C 180,E1 -8958.743,E2 -8958.743} C_VEL
LIN {X 0,Y 439.362,Z 172.755,A -85,B 0,C 180,E1 -8961.61,E2 -8961.61} C_VEL
LIN {X 0,Y 439.393,Z 172.753,A -85,B 0,C 180,E1 -8964.843,E2 -8964.843} C_VEL
LIN {X 0,Y 439.373,Z 172.756,A -85,B 0,C 180,E1 -8968.139,E2 -8968.139} C_VEL
LIN {X 0,Y 439.434,Z 172.746,A -85,B 0,C 180,E1 -8971.598,E2 -8971.598} C_VEL
LIN {X 0,Y 439.399,Z 172.754,A -85,B 0,C 180,E1 -8974.415,E2 -8974.415} C_VEL
LIN {X 0,Y 439.365,Z 172.754,A -85,B 0,C 180,E1 -8977.424,E2 -8977.424} C_VEL
LIN {X 0,Y 439.442,Z 172.746,A -85,B 0,C 180,E1 -8980.663,E2 -8980.663} C_VEL
LIN {X 0,Y 439.464,Z 172.746,A -85,B 0,C 180,E1 -8984.224,E2 -8984.224} C_VEL
LIN {X 0,Y 439.484,Z 172.743,A -85,B 0,C 180,E1 -8988.001,E2 -8988.001} C_VEL
LIN {X 0,Y 439.502,Z 172.74,A -85,B 0,C 180,E1 -8991.725,E2 -8991.725} C_VEL
LIN {X 0,Y 439.601,Z 172.725,A -85,B 0,C 180,E1 -8994.495,E2 -8994.495} C_VEL
LIN {X 0,Y 439.635,Z 172.721,A -85,B 0,C 180,E1 -8998.168,E2 -8998.168} C_VEL
LIN {X 0,Y 439.765,Z 172.705,A -85,B 0,C 180,E1 -9000,E2 -9000} C_VEL
LIN {X 0,Y 439.639,Z 172.722,A -85,B 0,C 180,E1 -9002.749,E2 -9002.749} C_VEL
LIN {X 0,Y 439.563,Z 172.73,A -85,B 0,C 180,E1 -9006.426,E2 -9006.426} C_VEL
LIN {X 0,Y 439.491,Z 172.74,A -85,B 0,C 180,E1 -9009.202,E2 -9009.202} C_VEL
LIN {X 0,Y 439.505,Z 172.739,A -85,B 0,C 180,E1 -9012.726,E2 -9012.726} C_VEL
LIN {X 0,Y 439.447,Z 172.746,A -85,B 0,C 180,E1 -9016.348,E2 -9016.348} C_VEL
LIN {X 0,Y 439.403,Z 172.75,A -85,B 0,C 180,E1 -9019.626,E2 -9019.626} C_VEL
LIN {X 0,Y 439.365,Z 172.756,A -85,B 0,C 180,E1 -9022.575,E2 -9022.575} C_VEL
LIN {X 0,Y 439.398,Z 172.751,A -85,B 0,C 180,E1 -9025.585,E2 -9025.585} C_VEL
LIN {X 0,Y 439.418,Z 172.749,A -85,B 0,C 180,E1 -9028.673,E2 -9028.673} C_VEL
LIN {X 0,Y 439.371,Z 172.757,A -85,B 0,C 180,E1 -9032.03,E2 -9032.03} C_VEL
LIN {X 0,Y 439.39,Z 172.753,A -85,B 0,C 180,E1 -9035.339,E2 -9035.339} C_VEL
LIN {X 0,Y 439.357,Z 172.754,A -85,B 0,C 180,E1 -9038.598,E2 -9038.598} C_VEL
LIN {X 0,Y 439.389,Z 172.756,A -85,B 0,C 180,E1 -9041.257,E2 -9041.257} C_VEL
LIN {X 0,Y 439.4,Z 172.753,A -85,B 0,C 180,E1 -9044.73,E2 -9044.73} C_VEL
LIN {X 0,Y 439.397,Z 172.75,A -85,B 0,C 180,E1 -9047.796,E2 -9047.796} C_VEL
LIN {X 0,Y 439.46,Z 172.944,A -85,B 0,C 180,E1 -9049.924,E2 -9049.924} C_VEL
LIN {X 0,Y 440.346,Z 178.481,A -85,B 0,C 180,E1 -9052.941,E2 -9052.941} C_VEL
LIN {X 0,Y 440.588,Z 182.405,A -85,B 0,C 180,E1 -9054.953,E2 -9054.953} C_VEL
LIN {X 0,Y 440.227,Z 189.117,A -85,B 0,C 180,E1 -9058.209,E2 -9058.209} C_VEL
LIN {X 0,Y 439.849,Z 196.162,A -85,B 0,C 180,E1 -9061.498,E2 -9061.498} C_VEL
LIN {X 0,Y 439.533,Z 202.616,A -85,B 0,C 180,E1 -9064.423,E2 -9064.423} C_VEL
LIN {X 0,Y 439.261,Z 209.353,A -85,B 0,C 180,E1 -9067.419,E2 -9067.419} C_VEL
LIN {X 0,Y 439.008,Z 217.145,A -85,B 0,C 180,E1 -9070.826,E2 -9070.826} C_VEL
LIN {X 0,Y 438.802,Z 223.476,A -85,B 0,C 180,E1 -9073.563,E2 -9073.563} C_VEL
LIN {X 0,Y 441.558,Z 239.287,A -85,B 0,C 180,E1 -9074.158,E2 -9074.158} C_VEL
LIN {X 0,Y 442.541,Z 247.978,A -85,B 0,C 180,E1 -9074.573,E2 -9074.573} C_VEL
LIN {X 0,Y 441.906,Z 260.193,A -85,B 0,C 180,E1 -9075.258,E2 -9075.258} C_VEL
LIN {X 0,Y 441.199,Z 272.646,A -85,B 0,C 180,E1 -9076.176,E2 -9076.176} C_VEL
LIN {X 0,Y 440.609,Z 283.562,A -85,B 0,C 180,E1 -9077.214,E2 -9077.214} C_VEL
LIN {X 0,Y 440.078,Z 292.464,A -85,B 0,C 180,E1 -9078.251,E2 -9078.251} C_VEL
LIN {X 0,Y 439.564,Z 300.646,A -85,B 0,C 180,E1 -9079.405,E2 -9079.405} C_VEL
LIN {X 0,Y 439.098,Z 308.676,A -85,B 0,C 180,E1 -9080.79,E2 -9080.79} C_VEL
LIN {X 0,Y 438.712,Z 315.115,A -85,B 0,C 180,E1 -9082.174,E2 -9082.174} C_VEL
LIN {X 0,Y 438.477,Z 321.181,A -85,B 0,C 180,E1 -9083.864,E2 -9083.864} C_VEL
LIN {X 0,Y 438.357,Z 325.276,A -85,B 0,C 180,E1 -9085.402,E2 -9085.402} C_VEL
LIN {X 0,Y 438.289,Z 327.138,A -85,B 0,C 180,E1 -9086.322,E2 -9086.322} C_VEL
LIN {X 0,Y 438.332,Z 328.537,A -85,B 0,C 180,E1 -9087.243,E2 -9087.243} C_VEL
LIN {X 0,Y 438.23,Z 330.141,A -85,B 0,C 180,E1 -9089.081,E2 -9089.081} C_VEL
LIN {X 0,Y 438.205,Z 330.357,A -85,B 0,C 180,E1 -9090,E2 -9090} C_VEL
LIN {X 0,Y 438.23,Z 330.142,A -85,B 0,C 180,E1 -9090.919,E2 -9090.919} C_VEL
LIN {X 0,Y 438.332,Z 328.541,A -85,B 0,C 180,E1 -9092.757,E2 -9092.757} C_VEL
LIN {X 0,Y 438.289,Z 327.143,A -85,B 0,C 180,E1 -9093.677,E2 -9093.677} C_VEL
LIN {X 0,Y 438.415,Z 324.207,A -85,B 0,C 180,E1 -9095.058,E2 -9095.058} C_VEL
LIN {X 0,Y 438.506,Z 320.231,A -85,B 0,C 180,E1 -9096.441,E2 -9096.441} C_VEL
LIN {X 0,Y 438.754,Z 314.118,A -85,B 0,C 180,E1 -9098.057,E2 -9098.057} C_VEL
LIN {X 0,Y 439.165,Z 307.442,A -85,B 0,C 180,E1 -9099.441,E2 -9099.441} C_VEL
LIN {X 0,Y 439.624,Z 299.156,A -85,B 0,C 180,E1 -9100.826,E2 -9100.826} C_VEL
LIN {X 0,Y 440.196,Z 290.668,A -85,B 0,C 180,E1 -9101.979,E2 -9101.979} C_VEL
LIN {X 0,Y 440.782,Z 281.117,A -85,B 0,C 180,E1 -9103.039,E2 -9103.039} C_VEL
LIN {X 0,Y 441.348,Z 269.8,A -85,B 0,C 180,E1 -9104.054,E2 -9104.054} C_VEL
LIN {X 0,Y 441.995,Z 258.429,A -85,B 0,C 180,E1 -9104.856,E2 -9104.856} C_VEL
LIN {X 0,Y 442.535,Z 246.767,A -85,B 0,C 180,E1 -9105.486,E2 -9105.486} C_VEL
LIN {X 0,Y 440.742,Z 234.672,A -85,B 0,C 180,E1 -9106.039,E2 -9106.039} C_VEL
LIN {X 0,Y 438.801,Z 223.477,A -85,B 0,C 180,E1 -9106.437,E2 -9106.437} C_VEL
LIN {X 0,Y 439.025,Z 216.068,A -85,B 0,C 180,E1 -9109.643,E2 -9109.643} C_VEL
LIN {X 0,Y 439.306,Z 208.241,A -85,B 0,C 180,E1 -9113.076,E2 -9113.076} C_VEL
LIN {X 0,Y 439.655,Z 200.356,A -85,B 0,C 180,E1 -9116.589,E2 -9116.589} C_VEL
LIN {X 0,Y 440.011,Z 193.598,A -85,B 0,C 180,E1 -9119.679,E2 -9119.679} C_VEL
LIN {X 0,Y 440.328,Z 186.87,A -85,B 0,C 180,E1 -9122.865,E2 -9122.865} C_VEL
LIN {X 0,Y 440.613,Z 181.361,A -85,B 0,C 180,E1 -9125.563,E2 -9125.563} C_VEL
LIN {X 0,Y 440.121,Z 176.887,A -85,B 0,C 180,E1 -9127.908,E2 -9127.908} C_VEL
LIN {X 0,Y 439.426,Z 172.754,A -85,B 0,C 180,E1 -9130.227,E2 -9130.227} C_VEL
LIN {X 0,Y 439.35,Z 172.76,A -85,B 0,C 180,E1 -9133.459,E2 -9133.459} C_VEL
LIN {X 0,Y 439.363,Z 172.756,A -85,B 0,C 180,E1 -9136.039,E2 -9136.039} C_VEL
LIN {X 0,Y 439.379,Z 172.754,A -85,B 0,C 180,E1 -9139.019,E2 -9139.019} C_VEL
LIN {X 0,Y 439.358,Z 172.754,A -85,B 0,C 180,E1 -9141.61,E2 -9141.61} C_VEL
LIN {X 0,Y 439.393,Z 172.752,A -85,B 0,C 180,E1 -9144.843,E2 -9144.843} C_VEL
LIN {X 0,Y 439.371,Z 172.756,A -85,B 0,C 180,E1 -9148.139,E2 -9148.139} C_VEL
LIN {X 0,Y 439.431,Z 172.748,A -85,B 0,C 180,E1 -9151.598,E2 -9151.598} C_VEL
LIN {X 0,Y 439.396,Z 172.752,A -85,B 0,C 180,E1 -9154.414,E2 -9154.414} C_VEL
LIN {X 0,Y 439.362,Z 172.756,A -85,B 0,C 180,E1 -9157.424,E2 -9157.424} C_VEL
LIN {X 0,Y 439.439,Z 172.745,A -85,B 0,C 180,E1 -9160.663,E2 -9160.663} C_VEL
LIN {X 0,Y 439.46,Z 172.744,A -85,B 0,C 180,E1 -9164.224,E2 -9164.224} C_VEL
LIN {X 0,Y 439.48,Z 172.741,A -85,B 0,C 180,E1 -9168.001,E2 -9168.001} C_VEL
LIN {X 0,Y 439.498,Z 172.738,A -85,B 0,C 180,E1 -9171.725,E2 -9171.725} C_VEL
LIN {X 0,Y 439.6,Z 172.725,A -85,B 0,C 180,E1 -9174.496,E2 -9174.496} C_VEL
LIN {X 0,Y 439.632,Z 172.722,A -85,B 0,C 180,E1 -9178.168,E2 -9178.168} C_VEL
LIN {X 0,Y 439.762,Z 172.706,A -85,B 0,C 180,E1 -9180,E2 -9180} C_VEL
LIN {X 0,Y 439.636,Z 172.723,A -85,B 0,C 180,E1 -9182.749,E2 -9182.749} C_VEL
LIN {X 0,Y 439.56,Z 172.733,A -85,B 0,C 180,E1 -9186.426,E2 -9186.426} C_VEL
LIN {X 0,Y 439.487,Z 172.738,A -85,B 0,C 180,E1 -9189.202,E2 -9189.202} C_VEL
LIN {X 0,Y 439.463,Z 172.743,A -85,B 0,C 180,E1 -9192.938,E2 -9192.938} C_VEL
LIN {X 0,Y 439.445,Z 172.747,A -85,B 0,C 180,E1 -9196.349,E2 -9196.349} C_VEL
LIN {X 0,Y 439.401,Z 172.752,A -85,B 0,C 180,E1 -9199.626,E2 -9199.626} C_VEL
LIN {X 0,Y 439.362,Z 172.755,A -85,B 0,C 180,E1 -9202.576,E2 -9202.576} C_VEL
LIN {X 0,Y 439.396,Z 172.753,A -85,B 0,C 180,E1 -9205.586,E2 -9205.586} C_VEL
LIN {X 0,Y 439.416,Z 172.748,A -85,B 0,C 180,E1 -9208.674,E2 -9208.674} C_VEL
LIN {X 0,Y 439.368,Z 172.756,A -85,B 0,C 180,E1 -9212.031,E2 -9212.031} C_VEL
LIN {X 0,Y 439.388,Z 172.754,A -85,B 0,C 180,E1 -9215.34,E2 -9215.34} C_VEL
LIN {X 0,Y 439.361,Z 172.755,A -85,B 0,C 180,E1 -9218.597,E2 -9218.597} C_VEL
LIN {X 0,Y 439.387,Z 172.755,A -85,B 0,C 180,E1 -9221.257,E2 -9221.257} C_VEL
LIN {X 0,Y 439.4,Z 172.754,A -85,B 0,C 180,E1 -9224.73,E2 -9224.73} C_VEL
LIN {X 0,Y 439.396,Z 172.751,A -85,B 0,C 180,E1 -9227.796,E2 -9227.796} C_VEL
LIN {X 0,Y 439.388,Z 172.754,A -85,B 0,C 180,E1 -9230.224,E2 -9230.224} C_VEL
LIN {X 0,Y 439.327,Z 172.765,A -85,B 0,C 180,E1 -9233.117,E2 -9233.117} C_VEL
LIN {X 0,Y 439.284,Z 173.243,A -85,B 0,C 180,E1 -9234.681,E2 -9234.681} C_VEL
LIN {X 0,Y 439.205,Z 176.295,A -85,B 0,C 180,E1 -9237.04,E2 -9237.04} C_VEL
LIN {X 0,Y 439.12,Z 180.568,A -85,B 0,C 180,E1 -9240.255,E2 -9240.255} C_VEL
LIN {X 0,Y 438.971,Z 185.271,A -85,B 0,C 180,E1 -9243.711,E2 -9243.711} C_VEL
LIN {X 0,Y 438.843,Z 189.019,A -85,B 0,C 180,E1 -9246.399,E2 -9246.399} C_VEL
LIN {X 0,Y 438.704,Z 193.296,A -85,B 0,C 180,E1 -9249.364,E2 -9249.364} C_VEL
LIN {X 0,Y 438.578,Z 197.646,A -85,B 0,C 180,E1 -9252.274,E2 -9252.274} C_VEL
LIN {X 0,Y 438.572,Z 199.757,A -85,B 0,C 180,E1 -9253.651,E2 -9253.651} C_VEL
LIN {X 0,Y 441.548,Z 213.224,A -85,B 0,C 180,E1 -9254.183,E2 -9254.183} C_VEL
LIN {X 0,Y 442.8,Z 221.419,A -85,B 0,C 180,E1 -9254.583,E2 -9254.583} C_VEL
LIN {X 0,Y 442.164,Z 233.836,A -85,B 0,C 180,E1 -9255.267,E2 -9255.267} C_VEL
LIN {X 0,Y 441.528,Z 246.365,A -85,B 0,C 180,E1 -9256.187,E2 -9256.187} C_VEL
LIN {X 0,Y 441.01,Z 257.334,A -85,B 0,C 180,E1 -9257.226,E2 -9257.226} C_VEL
LIN {X 0,Y 440.392,Z 266.24,A -85,B 0,C 180,E1 -9258.26,E2 -9258.26} C_VEL
LIN {X 0,Y 439.822,Z 275.884,A -85,B 0,C 180,E1 -9259.644,E2 -9259.644} C_VEL
LIN {X 0,Y 439.287,Z 283.58,A -85,B 0,C 180,E1 -9261.026,E2 -9261.026} C_VEL
LIN {X 0,Y 438.86,Z 290.639,A -85,B 0,C 180,E1 -9262.64,E2 -9262.64} C_VEL
LIN {X 0,Y 438.778,Z 292.081,A -85,B 0,C 180,E1 -9263.032,E2 -9263.032} C_VEL
LIN {X 0,Y 437.998,Z 294.517,A -85,B 0,C 180,E1 -9263.727,E2 -9263.727} C_VEL
LIN {X 0,Y 434.984,Z 297.94,A -85,B 0,C 180,E1 -9264.883,E2 -9264.883} C_VEL
LIN {X 0,Y 432.488,Z 300.159,A -85,B 0,C 180,E1 -9265.84,E2 -9265.84} C_VEL
LIN {X 0,Y 431.42,Z 301.532,A -85,B 0,C 180,E1 -9266.593,E2 -9266.593} C_VEL
LIN {X 0,Y 431.333,Z 301.891,A -85,B 0,C 180,E1 -9266.849,E2 -9266.849} C_VEL
LIN {X 0,Y 431.227,Z 303.412,A -85,B 0,C 180,E1 -9268.132,E2 -9268.132} C_VEL
LIN {X 0,Y 431.169,Z 304.262,A -85,B 0,C 180,E1 -9270,E2 -9270} C_VEL
LIN {X 0,Y 431.173,Z 304.074,A -85,B 0,C 180,E1 -9270.934,E2 -9270.934} C_VEL
LIN {X 0,Y 431.337,Z 302.522,A -85,B 0,C 180,E1 -9272.802,E2 -9272.802} C_VEL
LIN {X 0,Y 431.361,Z 301.169,A -85,B 0,C 180,E1 -9273.737,E2 -9273.737} C_VEL
LIN {X 0,Y 431.433,Z 298.307,A -85,B 0,C 180,E1 -9275.14,E2 -9275.14} C_VEL
LIN {X 0,Y 431.707,Z 293.75,A -85,B 0,C 180,E1 -9276.755,E2 -9276.755} C_VEL
LIN {X 0,Y 432.026,Z 287.443,A -85,B 0,C 180,E1 -9278.419,E2 -9278.419} C_VEL
LIN {X 0,Y 432.478,Z 280.659,A -85,B 0,C 180,E1 -9279.825,E2 -9279.825} C_VEL
LIN {X 0,Y 433.057,Z 272.186,A -85,B 0,C 180,E1 -9281.23,E2 -9281.23} C_VEL
LIN {X 0,Y 433.676,Z 263.469,A -85,B 0,C 180,E1 -9282.4,E2 -9282.4} C_VEL
LIN {X 0,Y 434.386,Z 252.506,A -85,B 0,C 180,E1 -9283.591,E2 -9283.591} C_VEL
LIN {X 0,Y 434.909,Z 241.965,A -85,B 0,C 180,E1 -9284.506,E2 -9284.506} C_VEL
LIN {X 0,Y 435.606,Z 229.869,A -85,B 0,C 180,E1 -9285.319,E2 -9285.319} C_VEL
LIN {X 0,Y 435.918,Z 221.1,A -85,B 0,C 180,E1 -9285.787,E2 -9285.787} C_VEL
LIN {X 0,Y 433.453,Z 208.398,A -85,B 0,C 180,E1 -9286.399,E2 -9286.399} C_VEL
LIN {X 0,Y 431.482,Z 199.936,A -85,B 0,C 180,E1 -9286.743,E2 -9286.743} C_VEL
LIN {X 0,Y 431.598,Z 195.077,A -85,B 0,C 180,E1 -9289.996,E2 -9289.996} C_VEL
LIN {X 0,Y 431.728,Z 190.766,A -85,B 0,C 180,E1 -9292.998,E2 -9292.998} C_VEL
LIN {X 0,Y 431.854,Z 186.512,A -85,B 0,C 180,E1 -9296.066,E2 -9296.066} C_VEL
LIN {X 0,Y 432.041,Z 182.278,A -85,B 0,C 180,E1 -9299.21,E2 -9299.21} C_VEL
LIN {X 0,Y 432.161,Z 177.987,A -85,B 0,C 180,E1 -9302.457,E2 -9302.457} C_VEL
LIN {X 0,Y 432.247,Z 175.115,A -85,B 0,C 180,E1 -9304.686,E2 -9304.686} C_VEL
LIN {X 0,Y 432.227,Z 173.679,A -85,B 0,C 180,E1 -9305.828,E2 -9305.828} C_VEL
LIN {X 0,Y 432.319,Z 173.633,A -85,B 0,C 180,E1 -9308.711,E2 -9308.711} C_VEL
LIN {X 0,Y 432.31,Z 173.635,A -85,B 0,C 180,E1 -9311.8,E2 -9311.8} C_VEL
LIN {X 0,Y 432.335,Z 173.63,A -85,B 0,C 180,E1 -9314.347,E2 -9314.347} C_VEL
LIN {X 0,Y 432.322,Z 173.635,A -85,B 0,C 180,E1 -9317.016,E2 -9317.016} C_VEL
LIN {X 0,Y 432.316,Z 173.631,A -85,B 0,C 180,E1 -9319.824,E2 -9319.824} C_VEL
LIN {X 0,Y 432.297,Z 173.637,A -85,B 0,C 180,E1 -9323.021,E2 -9323.021} C_VEL
LIN {X 0,Y 432.333,Z 173.632,A -85,B 0,C 180,E1 -9326.002,E2 -9326.002} C_VEL
LIN {X 0,Y 432.349,Z 173.628,A -85,B 0,C 180,E1 -9329.49,E2 -9329.49} C_VEL
LIN {X 0,Y 432.392,Z 173.623,A -85,B 0,C 180,E1 -9332.928,E2 -9332.928} C_VEL
LIN {X 0,Y 432.369,Z 173.629,A -85,B 0,C 180,E1 -9336.023,E2 -9336.023} C_VEL
LIN {X 0,Y 432.351,Z 173.628,A -85,B 0,C 180,E1 -9339.046,E2 -9339.046} C_VEL
LIN {X 0,Y 432.375,Z 173.628,A -85,B 0,C 180,E1 -9342.011,E2 -9342.011} C_VEL
LIN {X 0,Y 432.396,Z 173.623,A -85,B 0,C 180,E1 -9344.926,E2 -9344.926} C_VEL
LIN {X 0,Y 432.46,Z 173.619,A -85,B 0,C 180,E1 -9347.803,E2 -9347.803} C_VEL
LIN {X 0,Y 432.462,Z 173.618,A -85,B 0,C 180,E1 -9351.59,E2 -9351.59} C_VEL
LIN {X 0,Y 432.575,Z 173.6,A -85,B 0,C 180,E1 -9354.406,E2 -9354.406} C_VEL
LIN {X 0,Y 432.604,Z 173.597,A -85,B 0,C 180,E1 -9358.138,E2 -9358.138} C_VEL
LIN {X 0,Y 432.735,Z 173.581,A -85,B 0,C 180,E1 -9360,E2 -9360} C_VEL
LIN {X 0,Y 432.591,Z 173.6,A -85,B 0,C 180,E1 -9362.794,E2 -9362.794} C_VEL
LIN {X 0,Y 432.577,Z 173.599,A -85,B 0,C 180,E1 -9365.594,E2 -9365.594} C_VEL
LIN {X 0,Y 432.462,Z 173.615,A -85,B 0,C 180,E1 -9368.41,E2 -9368.41} C_VEL
LIN {X 0,Y 432.481,Z 173.614,A -85,B 0,C 180,E1 -9372.196,E2 -9372.196} C_VEL
LIN {X 0,Y 432.431,Z 173.621,A -85,B 0,C 180,E1 -9376.039,E2 -9376.039} C_VEL
LIN {X 0,Y 432.387,Z 173.623,A -85,B 0,C 180,E1 -9379.485,E2 -9379.485} C_VEL
LIN {X 0,Y 432.318,Z 173.631,A -85,B 0,C 180,E1 -9382.964,E2 -9382.964} C_VEL
LIN {X 0,Y 432.362,Z 173.631,A -85,B 0,C 180,E1 -9386.033,E2 -9386.033} C_VEL
LIN {X 0,Y 432.344,Z 173.63,A -85,B 0,C 180,E1 -9389.187,E2 -9389.187} C_VEL
LIN {X 0,Y 432.324,Z 173.633,A -85,B 0,C 180,E1 -9392.443,E2 -9392.443} C_VEL
LIN {X 0,Y 432.341,Z 173.633,A -85,B 0,C 180,E1 -9395.631,E2 -9395.631} C_VEL
LIN {X 0,Y 432.321,Z 173.63,A -85,B 0,C 180,E1 -9398.711,E2 -9398.711} C_VEL
LIN {X 0,Y 432.334,Z 173.631,A -85,B 0,C 180,E1 -9401.797,E2 -9401.797} C_VEL
LIN {X 0,Y 432.335,Z 173.634,A -85,B 0,C 180,E1 -9404.347,E2 -9404.347} C_VEL
LIN {X 0,Y 432.321,Z 173.632,A -85,B 0,C 180,E1 -9407.016,E2 -9407.016} C_VEL
LIN {X 0,Y 432.398,Z 173.817,A -85,B 0,C 180,E1 -9409.668,E2 -9409.668} C_VEL
LIN {X 0,Y 433.278,Z 179.158,A -85,B 0,C 180,E1 -9412.637,E2 -9412.637} C_VEL
LIN {X 0,Y 433.582,Z 183.418,A -85,B 0,C 180,E1 -9414.87,E2 -9414.87} C_VEL
LIN {X 0,Y 433.215,Z 190.116,A -85,B 0,C 180,E1 -9418.18,E2 -9418.18} C_VEL
LIN {X 0,Y 432.849,Z 196.583,A -85,B 0,C 180,E1 -9421.256,E2 -9421.256} C_VEL
LIN {X 0,Y 432.492,Z 203.596,A -85,B 0,C 180,E1 -9424.493,E2 -9424.493} C_VEL
LIN {X 0,Y 432.179,Z 210.319,A -85,B 0,C 180,E1 -9427.533,E2 -9427.533} C_VEL
LIN {X 0,Y 431.933,Z 217.379,A -85,B 0,C 180,E1 -9430.687,E2 -9430.687} C_VEL
LIN {X 0,Y 431.743,Z 223.453,A -85,B 0,C 180,E1 -9433.312,E2 -9433.312} C_VEL
LIN {X 0,Y 434.094,Z 236.8,A -85,B 0,C 180,E1 -9433.789,E2 -9433.789} C_VEL
LIN {X 0,Y 435.672,Z 247.764,A -85,B 0,C 180,E1 -9434.324,E2 -9434.324} C_VEL
LIN {X 0,Y 435.039,Z 259.98,A -85,B 0,C 180,E1 -9435.02,E2 -9435.02} C_VEL
LIN {X 0,Y 434.285,Z 272.432,A -85,B 0,C 180,E1 -9435.951,E2 -9435.951} C_VEL
LIN {X 0,Y 433.651,Z 283.347,A -85,B 0,C 180,E1 -9437.005,E2 -9437.005} C_VEL
LIN {X 0,Y 433.091,Z 292.25,A -85,B 0,C 180,E1 -9438.059,E2 -9438.059} C_VEL
LIN {X 0,Y 432.53,Z 300.431,A -85,B 0,C 180,E1 -9439.23,E2 -9439.23} C_VEL
LIN {X 0,Y 432.065,Z 308.462,A -85,B 0,C 180,E1 -9440.638,E2 -9440.638} C_VEL
LIN {X 0,Y 431.636,Z 314.901,A -85,B 0,C 180,E1 -9442.045,E2 -9442.045} C_VEL
LIN {X 0,Y 431.436,Z 320.332,A -85,B 0,C 180,E1 -9443.555,E2 -9443.555} C_VEL
LIN {X 0,Y 431.288,Z 325.063,A -85,B 0,C 180,E1 -9445.326,E2 -9445.326} C_VEL
LIN {X 0,Y 431.196,Z 326.925,A -85,B 0,C 180,E1 -9446.262,E2 -9446.262} C_VEL
LIN {X 0,Y 431.228,Z 328.324,A -85,B 0,C 180,E1 -9447.197,E2 -9447.197} C_VEL
LIN {X 0,Y 431.199,Z 329.321,A -85,B 0,C 180,E1 -9448.132,E2 -9448.132} C_VEL
LIN {X 0,Y 431.148,Z 329.928,A -85,B 0,C 180,E1 -9449.066,E2 -9449.066} C_VEL
LIN {X 0,Y 431.122,Z 330.145,A -85,B 0,C 180,E1 -9450,E2 -9450} C_VEL
LIN {X 0,Y 431.148,Z 329.929,A -85,B 0,C 180,E1 -9450.934,E2 -9450.934} C_VEL
LIN {X 0,Y 431.199,Z 329.323,A -85,B 0,C 180,E1 -9451.868,E2 -9451.868} C_VEL
LIN {X 0,Y 431.228,Z 328.328,A -85,B 0,C 180,E1 -9452.802,E2 -9452.802} C_VEL
LIN {X 0,Y 431.196,Z 326.929,A -85,B 0,C 180,E1 -9453.738,E2 -9453.738} C_VEL
LIN {X 0,Y 431.33,Z 323.994,A -85,B 0,C 180,E1 -9455.141,E2 -9455.141} C_VEL
LIN {X 0,Y 431.441,Z 320.017,A -85,B 0,C 180,E1 -9456.547,E2 -9456.547} C_VEL
LIN {X 0,Y 431.716,Z 313.905,A -85,B 0,C 180,E1 -9458.189,E2 -9458.189} C_VEL
LIN {X 0,Y 432.137,Z 307.228,A -85,B 0,C 180,E1 -9459.596,E2 -9459.596} C_VEL
LIN {X 0,Y 432.618,Z 298.942,A -85,B 0,C 180,E1 -9461.004,E2 -9461.004} C_VEL
LIN {X 0,Y 433.232,Z 290.454,A -85,B 0,C 180,E1 -9462.174,E2 -9462.174} C_VEL
LIN {X 0,Y 433.871,Z 280.332,A -85,B 0,C 180,E1 -9463.308,E2 -9463.308} C_VEL
LIN {X 0,Y 434.448,Z 269.587,A -85,B 0,C 180,E1 -9464.282,E2 -9464.282} C_VEL
LIN {X 0,Y 435.116,Z 258.215,A -85,B 0,C 180,E1 -9465.097,E2 -9465.097} C_VEL
LIN {X 0,Y 435.61,Z 246.551,A -85,B 0,C 180,E1 -9465.738,E2 -9465.738} C_VEL
LIN {X 0,Y 433.522,Z 233.228,A -85,B 0,C 180,E1 -9466.353,E2 -9466.353} C_VEL
LIN {X 0,Y 431.735,Z 223.263,A -85,B 0,C 180,E1 -9466.71,E2 -9466.71} C_VEL
LIN {X 0,Y 431.98,Z 215.885,A -85,B 0,C 180,E1 -9469.977,E2 -9469.977} C_VEL
LIN {X 0,Y 432.297,Z 208.093,A -85,B 0,C 180,E1 -9473.472,E2 -9473.472} C_VEL
LIN {X 0,Y 432.621,Z 201.012,A -85,B 0,C 180,E1 -9476.685,E2 -9476.685} C_VEL
LIN {X 0,Y 433.014,Z 193.468,A -85,B 0,C 180,E1 -9480.208,E2 -9480.208} C_VEL
LIN {X 0,Y 433.272,Z 188.728,A -85,B 0,C 180,E1 -9482.49,E2 -9482.49} C_VEL
LIN {X 0,Y 433.579,Z 183.408,A -85,B 0,C 180,E1 -9485.129,E2 -9485.129} C_VEL
LIN {X 0,Y 433.278,Z 179.145,A -85,B 0,C 180,E1 -9487.363,E2 -9487.363} C_VEL
LIN {X 0,Y 432.368,Z 173.632,A -85,B 0,C 180,E1 -9490.445,E2 -9490.445} C_VEL
LIN {X 0,Y 432.316,Z 173.635,A -85,B 0,C 180,E1 -9493.061,E2 -9493.061} C_VEL
LIN {X 0,Y 432.332,Z 173.631,A -85,B 0,C 180,E1 -9495.664,E2 -9495.664} C_VEL
LIN {X 0,Y 432.331,Z 173.633,A -85,B 0,C 180,E1 -9498.398,E2 -9498.398} C_VEL
LIN {X 0,Y 432.323,Z 173.631,A -85,B 0,C 180,E1 -9501.848,E2 -9501.848} C_VEL
LIN {X 0,Y 432.335,Z 173.63,A -85,B 0,C 180,E1 -9505.322,E2 -9505.322} C_VEL
LIN {X 0,Y 432.319,Z 173.634,A -85,B 0,C 180,E1 -9508.654,E2 -9508.654} C_VEL
LIN {X 0,Y 432.38,Z 173.627,A -85,B 0,C 180,E1 -9511.876,E2 -9511.876} C_VEL
LIN {X 0,Y 432.344,Z 173.628,A -85,B 0,C 180,E1 -9514.998,E2 -9514.998} C_VEL
LIN {X 0,Y 432.355,Z 173.629,A -85,B 0,C 180,E1 -9518.046,E2 -9518.046} C_VEL
LIN {X 0,Y 432.384,Z 173.625,A -85,B 0,C 180,E1 -9521.029,E2 -9521.029} C_VEL
LIN {X 0,Y 432.429,Z 173.621,A -85,B 0,C 180,E1 -9523.961,E2 -9523.961} C_VEL
LIN {X 0,Y 432.456,Z 173.617,A -85,B 0,C 180,E1 -9527.803,E2 -9527.803} C_VEL
LIN {X 0,Y 432.459,Z 173.616,A -85,B 0,C 180,E1 -9531.59,E2 -9531.59} C_VEL
LIN {X 0,Y 432.574,Z 173.6,A -85,B 0,C 180,E1 -9534.406,E2 -9534.406} C_VEL
LIN {X 0,Y 432.602,Z 173.597,A -85,B 0,C 180,E1 -9538.138,E2 -9538.138} C_VEL
LIN {X 0,Y 432.732,Z 173.581,A -85,B 0,C 180,E1 -9540,E2 -9540} C_VEL
LIN {X 0,Y 432.588,Z 173.602,A -85,B 0,C 180,E1 -9542.794,E2 -9542.794} C_VEL
LIN {X 0,Y 432.573,Z 173.6,A -85,B 0,C 180,E1 -9545.594,E2 -9545.594} C_VEL
LIN {X 0,Y 432.459,Z 173.618,A -85,B 0,C 180,E1 -9548.41,E2 -9548.41} C_VEL
LIN {X 0,Y 432.457,Z 173.62,A -85,B 0,C 180,E1 -9552.197,E2 -9552.197} C_VEL
LIN {X 0,Y 432.429,Z 173.621,A -85,B 0,C 180,E1 -9556.039,E2 -9556.039} C_VEL
LIN {X 0,Y 432.385,Z 173.626,A -85,B 0,C 180,E1 -9559.485,E2 -9559.485} C_VEL
LIN {X 0,Y 432.316,Z 173.632,A -85,B 0,C 180,E1 -9562.965,E2 -9562.965} C_VEL
LIN {X 0,Y 432.359,Z 173.629,A -85,B 0,C 180,E1 -9566.033,E2 -9566.033} C_VEL
LIN {X 0,Y 432.342,Z 173.631,A -85,B 0,C 180,E1 -9569.188,E2 -9569.188} C_VEL
LIN {X 0,Y 432.321,Z 173.632,A -85,B 0,C 180,E1 -9572.443,E2 -9572.443} C_VEL
LIN {X 0,Y 432.339,Z 173.633,A -85,B 0,C 180,E1 -9575.631,E2 -9575.631} C_VEL
LIN {X 0,Y 432.326,Z 173.632,A -85,B 0,C 180,E1 -9578.713,E2 -9578.713} C_VEL
LIN {X 0,Y 432.332,Z 173.63,A -85,B 0,C 180,E1 -9581.797,E2 -9581.797} C_VEL
LIN {X 0,Y 432.333,Z 173.631,A -85,B 0,C 180,E1 -9584.348,E2 -9584.348} C_VEL
LIN {X 0,Y 432.32,Z 173.634,A -85,B 0,C 180,E1 -9587.016,E2 -9587.016} C_VEL
LIN {X 0,Y 432.333,Z 173.631,A -85,B 0,C 180,E1 -9589.821,E2 -9589.821} C_VEL
LIN {X 0,Y 432.289,Z 173.641,A -85,B 0,C 180,E1 -9593.021,E2 -9593.021} C_VEL
LIN {X 0,Y 432.213,Z 173.826,A -85,B 0,C 180,E1 -9594.393,E2 -9594.393} C_VEL
LIN {X 0,Y 432.153,Z 177.843,A -85,B 0,C 180,E1 -9597.543,E2 -9597.543} C_VEL
LIN {X 0,Y 432.025,Z 182.113,A -85,B 0,C 180,E1 -9600.789,E2 -9600.789} C_VEL
LIN {X 0,Y 431.878,Z 186.361,A -85,B 0,C 180,E1 -9603.936,E2 -9603.936} C_VEL
LIN {X 0,Y 431.75,Z 190.616,A -85,B 0,C 180,E1 -9607.004,E2 -9607.004} C_VEL
LIN {X 0,Y 431.609,Z 194.926,A -85,B 0,C 180,E1 -9610.005,E2 -9610.005} C_VEL
LIN {X 0,Y 431.515,Z 200.049,A -85,B 0,C 180,E1 -9613.38,E2 -9613.38} C_VEL
LIN {X 0,Y 434.474,Z 213.381,A -85,B 0,C 180,E1 -9613.916,E2 -9613.916} C_VEL
LIN {X 0,Y 435.948,Z 221.643,A -85,B 0,C 180,E1 -9614.334,E2 -9614.334} C_VEL
LIN {X 0,Y 435.311,Z 234.056,A -85,B 0,C 180,E1 -9615.03,E2 -9615.03} C_VEL
LIN {X 0,Y 434.734,Z 245.163,A -85,B 0,C 180,E1 -9615.847,E2 -9615.847} C_VEL
LIN {X 0,Y 434.147,Z 256.476,A -85,B 0,C 180,E1 -9616.901,E2 -9616.901} C_VEL
LIN {X 0,Y 433.454,Z 266.456,A -85,B 0,C 180,E1 -9618.07,E2 -9618.07} C_VEL
LIN {X 0,Y 432.82,Z 276.1,A -85,B 0,C 180,E1 -9619.475,E2 -9619.475} C_VEL
LIN {X 0,Y 432.272,Z 283.795,A -85,B 0,C 180,E1 -9620.879,E2 -9620.879} C_VEL
LIN {X 0,Y 431.809,Z 290.854,A -85,B 0,C 180,E1 -9622.519,E2 -9622.519} C_VEL
LIN {X 0,Y 431.653,Z 295.553,A -85,B 0,C 180,E1 -9623.925,E2 -9623.925} C_VEL
LIN {X 0,Y 431.363,Z 299.156,A -85,B 0,C 180,E1 -9625.328,E2 -9625.328} C_VEL
LIN {X 0,Y 431.333,Z 301.891,A -85,B 0,C 180,E1 -9626.849,E2 -9626.849} C_VEL
LIN {X 0,Y 430.637,Z 302.94,A -85,B 0,C 180,E1 -9627.616,E2 -9627.616} C_VEL
LIN {X 0,Y 427.676,Z 304.037,A -85,B 0,C 180,E1 -9628.87,E2 -9628.87} C_VEL
LIN {X 0,Y 425.195,Z 304.423,A -85,B 0,C 180,E1 -9629.889,E2 -9629.889} C_VEL
LIN {X 0,Y 424.16,Z 304.375,A -85,B 0,C 180,E1 -9630.678,E2 -9630.678} C_VEL
LIN {X 0,Y 424.092,Z 304.288,A -85,B 0,C 180,E1 -9630.946,E2 -9630.946} C_VEL
LIN {X 0,Y 424.27,Z 302.734,A -85,B 0,C 180,E1 -9632.849,E2 -9632.849} C_VEL
LIN {X 0,Y 424.266,Z 301.381,A -85,B 0,C 180,E1 -9633.799,E2 -9633.799} C_VEL
LIN {X 0,Y 424.383,Z 298.518,A -85,B 0,C 180,E1 -9635.226,E2 -9635.226} C_VEL
LIN {X 0,Y 424.634,Z 294.312,A -85,B 0,C 180,E1 -9636.76,E2 -9636.76} C_VEL
LIN {X 0,Y 424.856,Z 289.626,A -85,B 0,C 180,E1 -9638.083,E2 -9638.083} C_VEL
LIN {X 0,Y 425.331,Z 283.317,A -85,B 0,C 180,E1 -9639.511,E2 -9639.511} C_VEL
LIN {X 0,Y 425.908,Z 275.418,A -85,B 0,C 180,E1 -9640.939,E2 -9640.939} C_VEL
LIN {X 0,Y 426.597,Z 265.592,A -85,B 0,C 180,E1 -9642.367,E2 -9642.367} C_VEL
LIN {X 0,Y 427.278,Z 256.041,A -85,B 0,C 180,E1 -9643.477,E2 -9643.477} C_VEL
LIN {X 0,Y 427.868,Z 245.065,A -85,B 0,C 180,E1 -9644.507,E2 -9644.507} C_VEL
LIN {X 0,Y 428.579,Z 233.883,A -85,B 0,C 180,E1 -9645.333,E2 -9645.333} C_VEL
LIN {X 0,Y 429.09,Z 222.542,A -85,B 0,C 180,E1 -9645.984,E2 -9645.984} C_VEL
LIN {X 0,Y 426.774,Z 210.146,A -85,B 0,C 180,E1 -9646.611,E2 -9646.611} C_VEL
LIN {X 0,Y 424.425,Z 200.15,A -85,B 0,C 180,E1 -9647.023,E2 -9647.023} C_VEL
LIN {X 0,Y 424.539,Z 195.266,A -85,B 0,C 180,E1 -9650.343,E2 -9650.343} C_VEL
LIN {X 0,Y 424.701,Z 190.938,A -85,B 0,C 180,E1 -9653.401,E2 -9653.401} C_VEL
LIN {X 0,Y 424.848,Z 186.429,A -85,B 0,C 180,E1 -9656.71,E2 -9656.71} C_VEL
LIN {X 0,Y 425.004,Z 182.418,A -85,B 0,C 180,E1 -9659.742,E2 -9659.742} C_VEL
LIN {X 0,Y 425.131,Z 178.117,A -85,B 0,C 180,E1 -9663.061,E2 -9663.061} C_VEL
LIN {X 0,Y 425.183,Z 174.538,A -85,B 0,C 180,E1 -9665.91,E2 -9665.91} C_VEL
LIN {X 0,Y 425.277,Z 174.511,A -85,B 0,C 180,E1 -9668.901,E2 -9668.901} C_VEL
LIN {X 0,Y 425.262,Z 174.513,A -85,B 0,C 180,E1 -9672.655,E2 -9672.655} C_VEL
LIN {X 0,Y 425.286,Z 174.512,A -85,B 0,C 180,E1 -9675.283,E2 -9675.283} C_VEL
LIN {X 0,Y 425.274,Z 174.511,A -85,B 0,C 180,E1 -9678.621,E2 -9678.621} C_VEL
LIN {X 0,Y 425.289,Z 174.51,A -85,B 0,C 180,E1 -9681.1,E2 -9681.1} C_VEL
LIN {X 0,Y 425.293,Z 174.51,A -85,B 0,C 180,E1 -9684.663,E2 -9684.663} C_VEL
LIN {X 0,Y 425.266,Z 174.513,A -85,B 0,C 180,E1 -9688.073,E2 -9688.073} C_VEL
LIN {X 0,Y 425.333,Z 174.502,A -85,B 0,C 180,E1 -9691.368,E2 -9691.368} C_VEL
LIN {X 0,Y 425.355,Z 174.499,A -85,B 0,C 180,E1 -9693.505,E2 -9693.505} C_VEL
LIN {X 0,Y 425.306,Z 174.506,A -85,B 0,C 180,E1 -9696.635,E2 -9696.635} C_VEL
LIN {X 0,Y 425.329,Z 174.505,A -85,B 0,C 180,E1 -9700.364,E2 -9700.364} C_VEL
LIN {X 0,Y 425.389,Z 174.498,A -85,B 0,C 180,E1 -9703.688,E2 -9703.688} C_VEL
LIN {X 0,Y 425.413,Z 174.495,A -85,B 0,C 180,E1 -9707.598,E2 -9707.598} C_VEL
LIN {X 0,Y 425.407,Z 174.497,A -85,B 0,C 180,E1 -9711.449,E2 -9711.449} C_VEL
LIN {X 0,Y 425.529,Z 174.477,A -85,B 0,C 180,E1 -9714.313,E2 -9714.313} C_VEL
LIN {X 0,Y 425.574,Z 174.473,A -85,B 0,C 180,E1 -9718.107,E2 -9718.107} C_VEL
LIN {X 0,Y 425.705,Z 174.456,A -85,B 0,C 180,E1 -9720,E2 -9720} C_VEL
LIN {X 0,Y 425.544,Z 174.478,A -85,B 0,C 180,E1 -9722.84,E2 -9722.84} C_VEL
LIN {X 0,Y 425.531,Z 174.477,A -85,B 0,C 180,E1 -9725.687,E2 -9725.687} C_VEL
LIN {X 0,Y 425.407,Z 174.495,A -85,B 0,C 180,E1 -9728.551,E2 -9728.551} C_VEL
LIN {X 0,Y 425.431,Z 174.494,A -85,B 0,C 180,E1 -9732.401,E2 -9732.401} C_VEL
LIN {X 0,Y 425.389,Z 174.498,A -85,B 0,C 180,E1 -9736.312,E2 -9736.312} C_VEL
LIN {X 0,Y 425.329,Z 174.503,A -85,B 0,C 180,E1 -9739.635,E2 -9739.635} C_VEL
LIN {X 0,Y 425.289,Z 174.512,A -85,B 0,C 180,E1 -9742.339,E2 -9742.339} C_VEL
LIN {X 0,Y 425.292,Z 174.507,A -85,B 0,C 180,E1 -9745.446,E2 -9745.446} C_VEL
LIN {X 0,Y 425.349,Z 174.502,A -85,B 0,C 180,E1 -9747.558,E2 -9747.558} C_VEL
LIN {X 0,Y 425.289,Z 174.508,A -85,B 0,C 180,E1 -9750.816,E2 -9750.816} C_VEL
LIN {X 0,Y 425.311,Z 174.506,A -85,B 0,C 180,E1 -9754.288,E2 -9754.288} C_VEL
LIN {X 0,Y 425.271,Z 174.514,A -85,B 0,C 180,E1 -9757.695,E2 -9757.695} C_VEL
LIN {X 0,Y 425.273,Z 174.514,A -85,B 0,C 180,E1 -9761.379,E2 -9761.379} C_VEL
LIN {X 0,Y 425.286,Z 174.511,A -85,B 0,C 180,E1 -9764.717,E2 -9764.717} C_VEL
LIN {X 0,Y 425.292,Z 174.508,A -85,B 0,C 180,E1 -9768.042,E2 -9768.042} C_VEL
LIN {X 0,Y 425.306,Z 174.555,A -85,B 0,C 180,E1 -9769.32,E2 -9769.32} C_VEL
LIN {X 0,Y 426.247,Z 179.963,A -85,B 0,C 180,E1 -9772.406,E2 -9772.406} C_VEL
LIN {X 0,Y 426.589,Z 184.424,A -85,B 0,C 180,E1 -9774.787,E2 -9774.787} C_VEL
LIN {X 0,Y 426.205,Z 191.11,A -85,B 0,C 180,E1 -9778.152,E2 -9778.152} C_VEL
LIN {X 0,Y 425.795,Z 197.833,A -85,B 0,C 180,E1 -9781.402,E2 -9781.402} C_VEL
LIN {X 0,Y 425.421,Z 204.575,A -85,B 0,C 180,E1 -9784.563,E2 -9784.563} C_VEL
LIN {X 0,Y 425.095,Z 211.582,A -85,B 0,C 180,E1 -9787.795,E2 -9787.795} C_VEL
LIN {X 0,Y 424.815,Z 219.029,A -85,B 0,C 180,E1 -9791.179,E2 -9791.179} C_VEL
LIN {X 0,Y 424.674,Z 223.047,A -85,B 0,C 180,E1 -9793,E2 -9793} C_VEL
LIN {X 0,Y 427.357,Z 238.525,A -85,B 0,C 180,E1 -9793.604,E2 -9793.604} C_VEL
LIN {X 0,Y 428.782,Z 248.682,A -85,B 0,C 180,E1 -9794.126,E2 -9794.126} C_VEL
LIN {X 0,Y 428.065,Z 261.535,A -85,B 0,C 180,E1 -9794.892,E2 -9794.892} C_VEL
LIN {X 0,Y 427.386,Z 272.218,A -85,B 0,C 180,E1 -9795.72,E2 -9795.72} C_VEL
LIN {X 0,Y 426.701,Z 283.133,A -85,B 0,C 180,E1 -9796.789,E2 -9796.789} C_VEL
LIN {X 0,Y 426.124,Z 292.036,A -85,B 0,C 180,E1 -9797.861,E2 -9797.861} C_VEL
LIN {X 0,Y 425.52,Z 300.217,A -85,B 0,C 180,E1 -9799.051,E2 -9799.051} C_VEL
LIN {X 0,Y 425.028,Z 308.248,A -85,B 0,C 180,E1 -9800.482,E2 -9800.482} C_VEL
LIN {X 0,Y 424.585,Z 314.687,A -85,B 0,C 180,E1 -9801.912,E2 -9801.912} C_VEL
LIN {X 0,Y 424.337,Z 320.536,A -85,B 0,C 180,E1 -9803.586,E2 -9803.586} C_VEL
LIN {X 0,Y 424.219,Z 324.85,A -85,B 0,C 180,E1 -9805.248,E2 -9805.248} C_VEL
LIN {X 0,Y 424.107,Z 326.712,A -85,B 0,C 180,E1 -9806.199,E2 -9806.199} C_VEL
LIN {X 0,Y 424.126,Z 328.111,A -85,B 0,C 180,E1 -9807.15,E2 -9807.15} C_VEL
LIN {X 0,Y 424.125,Z 329.108,A -85,B 0,C 180,E1 -9808.101,E2 -9808.101} C_VEL
LIN {X 0,Y 424.069,Z 329.716,A -85,B 0,C 180,E1 -9809.05,E2 -9809.05} C_VEL
LIN {X 0,Y 424.041,Z 329.932,A -85,B 0,C 180,E1 -9810,E2 -9810} C_VEL
LIN {X 0,Y 424.125,Z 329.111,A -85,B 0,C 180,E1 -9811.899,E2 -9811.899} C_VEL
LIN {X 0,Y 424.125,Z 328.114,A -85,B 0,C 180,E1 -9812.849,E2 -9812.849} C_VEL
LIN {X 0,Y 424.107,Z 326.716,A -85,B 0,C 180,E1 -9813.8,E2 -9813.8} C_VEL
LIN {X 0,Y 424.246,Z 323.78,A -85,B 0,C 180,E1 -9815.227,E2 -9815.227} C_VEL
LIN {X 0,Y 424.359,Z 319.803,A -85,B 0,C 180,E1 -9816.657,E2 -9816.657} C_VEL
LIN {X 0,Y 424.666,Z 313.691,A -85,B 0,C 180,E1 -9818.326,E2 -9818.326} C_VEL
LIN {X 0,Y 425.087,Z 307.013,A -85,B 0,C 180,E1 -9819.756,E2 -9819.756} C_VEL
LIN {X 0,Y 425.623,Z 298.728,A -85,B 0,C 180,E1 -9821.187,E2 -9821.187} C_VEL
LIN {X 0,Y 426.279,Z 290.24,A -85,B 0,C 180,E1 -9822.376,E2 -9822.376} C_VEL
LIN {X 0,Y 426.917,Z 280.543,A -85,B 0,C 180,E1 -9823.485,E2 -9823.485} C_VEL
LIN {X 0,Y 427.541,Z 269.373,A -85,B 0,C 180,E1 -9824.518,E2 -9824.518} C_VEL
LIN {X 0,Y 428.248,Z 258.001,A -85,B 0,C 180,E1 -9825.345,E2 -9825.345} C_VEL
LIN {X 0,Y 428.727,Z 247.547,A -85,B 0,C 180,E1 -9825.937,E2 -9825.937} C_VEL
LIN {X 0,Y 426.722,Z 234.366,A -85,B 0,C 180,E1 -9826.576,E2 -9826.576} C_VEL
LIN {X 0,Y 424.673,Z 223.048,A -85,B 0,C 180,E1 -9827,E2 -9827} C_VEL
LIN {X 0,Y 424.936,Z 215.72,A -85,B 0,C 180,E1 -9830.323,E2 -9830.323} C_VEL
LIN {X 0,Y 425.268,Z 207.936,A -85,B 0,C 180,E1 -9833.884,E2 -9833.884} C_VEL
LIN {X 0,Y 425.582,Z 201.411,A -85,B 0,C 180,E1 -9836.906,E2 -9836.906} C_VEL
LIN {X 0,Y 426.001,Z 194.455,A -85,B 0,C 180,E1 -9840.21,E2 -9840.21} C_VEL
LIN {X 0,Y 426.291,Z 188.865,A -85,B 0,C 180,E1 -9842.959,E2 -9842.959} C_VEL
LIN {X 0,Y 426.588,Z 184.413,A -85,B 0,C 180,E1 -9845.213,E2 -9845.213} C_VEL
LIN {X 0,Y 426.2,Z 179.812,A -85,B 0,C 180,E1 -9847.672,E2 -9847.672} C_VEL
LIN {X 0,Y 425.306,Z 174.511,A -85,B 0,C 180,E1 -9850.737,E2 -9850.737} C_VEL
LIN {X 0,Y 425.261,Z 174.516,A -85,B 0,C 180,E1 -9853.955,E2 -9853.955} C_VEL
LIN {X 0,Y 425.273,Z 174.51,A -85,B 0,C 180,E1 -9857.347,E2 -9857.347} C_VEL
LIN {X 0,Y 425.27,Z 174.51,A -85,B 0,C 180,E1 -9860.961,E2 -9860.961} C_VEL
LIN {X 0,Y 425.275,Z 174.512,A -85,B 0,C 180,E1 -9864.072,E2 -9864.072} C_VEL
LIN {X 0,Y 425.28,Z 174.509,A -85,B 0,C 180,E1 -9866.952,E2 -9866.952} C_VEL
LIN {X 0,Y 425.289,Z 174.511,A -85,B 0,C 180,E1 -9870.28,E2 -9870.28} C_VEL
LIN {X 0,Y 425.352,Z 174.501,A -85,B 0,C 180,E1 -9873.505,E2 -9873.505} C_VEL
LIN {X 0,Y 425.282,Z 174.507,A -85,B 0,C 180,E1 -9876.633,E2 -9876.633} C_VEL
LIN {X 0,Y 425.293,Z 174.511,A -85,B 0,C 180,E1 -9879.694,E2 -9879.694} C_VEL
LIN {X 0,Y 425.34,Z 174.501,A -85,B 0,C 180,E1 -9882.697,E2 -9882.697} C_VEL
LIN {X 0,Y 425.346,Z 174.504,A -85,B 0,C 180,E1 -9885.65,E2 -9885.65} C_VEL
LIN {X 0,Y 425.346,Z 174.501,A -85,B 0,C 180,E1 -9888.564,E2 -9888.564} C_VEL
LIN {X 0,Y 425.403,Z 174.496,A -85,B 0,C 180,E1 -9891.449,E2 -9891.449} C_VEL
LIN {X 0,Y 425.528,Z 174.477,A -85,B 0,C 180,E1 -9894.313,E2 -9894.313} C_VEL
LIN {X 0,Y 425.571,Z 174.473,A -85,B 0,C 180,E1 -9898.107,E2 -9898.107} C_VEL
LIN {X 0,Y 425.701,Z 174.457,A -85,B 0,C 180,E1 -9900,E2 -9900} C_VEL
LIN {X 0,Y 425.541,Z 174.48,A -85,B 0,C 180,E1 -9902.84,E2 -9902.84} C_VEL
LIN {X 0,Y 425.528,Z 174.478,A -85,B 0,C 180,E1 -9905.687,E2 -9905.687} C_VEL
LIN {X 0,Y 425.403,Z 174.498,A -85,B 0,C 180,E1 -9908.551,E2 -9908.551} C_VEL
LIN {X 0,Y 425.41,Z 174.496,A -85,B 0,C 180,E1 -9912.402,E2 -9912.402} C_VEL
LIN {X 0,Y 425.386,Z 174.498,A -85,B 0,C 180,E1 -9916.312,E2 -9916.312} C_VEL
LIN {X 0,Y 425.327,Z 174.505,A -85,B 0,C 180,E1 -9919.636,E2 -9919.636} C_VEL
LIN {X 0,Y 425.303,Z 174.507,A -85,B 0,C 180,E1 -9923.365,E2 -9923.365} C_VEL
LIN {X 0,Y 425.346,Z 174.5,A -85,B 0,C 180,E1 -9926.845,E2 -9926.845} C_VEL
LIN {X 0,Y 425.29,Z 174.51,A -85,B 0,C 180,E1 -9929.72,E2 -9929.72} C_VEL
LIN {X 0,Y 425.281,Z 174.511,A -85,B 0,C 180,E1 -9933.048,E2 -9933.048} C_VEL
LIN {X 0,Y 425.276,Z 174.51,A -85,B 0,C 180,E1 -9935.928,E2 -9935.928} C_VEL
LIN {X 0,Y 425.271,Z 174.513,A -85,B 0,C 180,E1 -9939.04,E2 -9939.04} C_VEL
LIN {X 0,Y 425.274,Z 174.511,A -85,B 0,C 180,E1 -9942.653,E2 -9942.653} C_VEL
LIN {X 0,Y 425.261,Z 174.511,A -85,B 0,C 180,E1 -9946.045,E2 -9946.045} C_VEL
LIN {X 0,Y 425.274,Z 174.513,A -85,B 0,C 180,E1 -9948.622,E2 -9948.622} C_VEL
LIN {X 0,Y 425.291,Z 174.51,A -85,B 0,C 180,E1 -9951.101,E2 -9951.101} C_VEL
LIN {X 0,Y 425.169,Z 174.527,A -85,B 0,C 180,E1 -9954.093,E2 -9954.093} C_VEL
LIN {X 0,Y 425.118,Z 177.974,A -85,B 0,C 180,E1 -9956.938,E2 -9956.938} C_VEL
LIN {X 0,Y 424.995,Z 182.263,A -85,B 0,C 180,E1 -9960.258,E2 -9960.258} C_VEL
LIN {X 0,Y 424.856,Z 186.528,A -85,B 0,C 180,E1 -9963.472,E2 -9963.472} C_VEL
LIN {X 0,Y 424.72,Z 190.793,A -85,B 0,C 180,E1 -9966.601,E2 -9966.601} C_VEL
LIN {X 0,Y 424.555,Z 195.118,A -85,B 0,C 180,E1 -9969.658,E2 -9969.658} C_VEL
LIN {X 0,Y 424.439,Z 200.158,A -85,B 0,C 180,E1 -9973.08,E2 -9973.08} C_VEL
LIN {X 0,Y 427.641,Z 214.44,A -85,B 0,C 180,E1 -9973.685,E2 -9973.685} C_VEL
LIN {X 0,Y 429.079,Z 223.036,A -85,B 0,C 180,E1 -9974.138,E2 -9974.138} C_VEL
LIN {X 0,Y 428.376,Z 236.038,A -85,B 0,C 180,E1 -9974.904,E2 -9974.904} C_VEL
LIN {X 0,Y 427.739,Z 247.485,A -85,B 0,C 180,E1 -9975.792,E2 -9975.792} C_VEL
LIN {X 0,Y 427.119,Z 258.833,A -85,B 0,C 180,E1 -9976.924,E2 -9976.924} C_VEL
LIN {X 0,Y 426.38,Z 268.446,A -85,B 0,C 180,E1 -9978.11,E2 -9978.11} C_VEL
LIN {X 0,Y 425.822,Z 276.317,A -85,B 0,C 180,E1 -9979.3,E2 -9979.3} C_VEL
LIN {X 0,Y 425.27,Z 284.01,A -85,B 0,C 180,E1 -9980.728,E2 -9980.728} C_VEL
LIN {X 0,Y 424.76,Z 291.069,A -85,B 0,C 180,E1 -9982.394,E2 -9982.394} C_VEL
LIN {X 0,Y 424.59,Z 295.767,A -85,B 0,C 180,E1 -9983.824,E2 -9983.824} C_VEL
LIN {X 0,Y 424.296,Z 299.37,A -85,B 0,C 180,E1 -9985.25,E2 -9985.25} C_VEL
LIN {X 0,Y 424.257,Z 302.175,A -85,B 0,C 180,E1 -9986.845,E2 -9986.845} C_VEL
LIN {X 0,Y 424.154,Z 303.625,A -85,B 0,C 180,E1 -9988.101,E2 -9988.101} C_VEL
LIN {X 0,Y 424.086,Z 304.474,A -85,B 0,C 180,E1 -9990,E2 -9990} C_VEL
LIN {X 0,Y 424.092,Z 304.288,A -85,B 0,C 180,E1 -9990.946,E2 -9990.946} C_VEL
LIN {X 0,Y 423.46,Z 303.97,A -85,B 0,C 180,E1 -9991.738,E2 -9991.738} C_VEL
LIN {X 0,Y 420.613,Z 302.791,A -85,B 0,C 180,E1 -9993.019,E2 -9993.019} C_VEL
LIN {X 0,Y 418.244,Z 301.272,A -85,B 0,C 180,E1 -9994.042,E2 -9994.042} C_VEL
LIN {X 0,Y 417.309,Z 299.805,A -85,B 0,C 180,E1 -9994.822,E2 -9994.822} C_VEL
LIN {X 0,Y 417.278,Z 299.237,A -85,B 0,C 180,E1 -9995.083,E2 -9995.083} C_VEL
LIN {X 0,Y 417.562,Z 294.846,A -85,B 0,C 180,E1 -9996.766,E2 -9996.766} C_VEL
LIN {X 0,Y 417.82,Z 289.837,A -85,B 0,C 180,E1 -9998.22,E2 -9998.22} C_VEL
LIN {X 0,Y 418.337,Z 283.527,A -85,B 0,C 180,E1 -9999.672,E2 -9999.672} C_VEL
LIN {X 0,Y 418.945,Z 275.628,A -85,B 0,C 180,E1 -10001.123,E2 -10001.123} C_VEL
LIN {X 0,Y 419.52,Z 267.576,A -85,B 0,C 180,E1 -10002.333,E2 -10002.333} C_VEL
LIN {X 0,Y 420.281,Z 257.746,A -85,B 0,C 180,E1 -10003.539,E2 -10003.539} C_VEL
LIN {X 0,Y 420.946,Z 246.693,A -85,B 0,C 180,E1 -10004.627,E2 -10004.627} C_VEL
LIN {X 0,Y 421.644,Z 235.85,A -85,B 0,C 180,E1 -10005.468,E2 -10005.468} C_VEL
LIN {X 0,Y 422.231,Z 223.978,A -85,B 0,C 180,E1 -10006.183,E2 -10006.183} C_VEL
LIN {X 0,Y 420.138,Z 212.081,A -85,B 0,C 180,E1 -10006.818,E2 -10006.818} C_VEL
LIN {X 0,Y 417.351,Z 200.351,A -85,B 0,C 180,E1 -10007.323,E2 -10007.323} C_VEL
LIN {X 0,Y 417.469,Z 196.904,A -85,B 0,C 180,E1 -10009.676,E2 -10009.676} C_VEL
LIN {X 0,Y 417.599,Z 192.569,A -85,B 0,C 180,E1 -10012.773,E2 -10012.773} C_VEL
LIN {X 0,Y 417.733,Z 188.256,A -85,B 0,C 180,E1 -10015.94,E2 -10015.94} C_VEL
LIN {X 0,Y 417.93,Z 183.993,A -85,B 0,C 180,E1 -10019.188,E2 -10019.188} C_VEL
LIN {X 0,Y 418.092,Z 179.683,A -85,B 0,C 180,E1 -10022.542,E2 -10022.542} C_VEL
LIN {X 0,Y 418.163,Z 176.795,A -85,B 0,C 180,E1 -10024.85,E2 -10024.85} C_VEL
LIN {X 0,Y 418.174,Z 175.398,A -85,B 0,C 180,E1 -10026.224,E2 -10026.224} C_VEL
LIN {X 0,Y 418.206,Z 175.393,A -85,B 0,C 180,E1 -10029.372,E2 -10029.372} C_VEL
LIN {X 0,Y 418.214,Z 175.389,A -85,B 0,C 180,E1 -10032.318,E2 -10032.318} C_VEL
LIN {X 0,Y 418.237,Z 175.39,A -85,B 0,C 180,E1 -10035.109,E2 -10035.109} C_VEL
LIN {X 0,Y 418.242,Z 175.385,A -85,B 0,C 180,E1 -10037.767,E2 -10037.767} C_VEL
LIN {X 0,Y 418.242,Z 175.385,A -85,B 0,C 180,E1 -10041.557,E2 -10041.557} C_VEL
LIN {X 0,Y 418.25,Z 175.386,A -85,B 0,C 180,E1 -10045.158,E2 -10045.158} C_VEL
LIN {X 0,Y 418.245,Z 175.385,A -85,B 0,C 180,E1 -10047.472,E2 -10047.472} C_VEL
LIN {X 0,Y 418.27,Z 175.384,A -85,B 0,C 180,E1 -10050.895,E2 -10050.895} C_VEL
LIN {X 0,Y 418.27,Z 175.385,A -85,B 0,C 180,E1 -10054.096,E2 -10054.096} C_VEL
LIN {X 0,Y 418.239,Z 175.385,A -85,B 0,C 180,E1 -10057.264,E2 -10057.264} C_VEL
LIN {X 0,Y 418.284,Z 175.383,A -85,B 0,C 180,E1 -10060.364,E2 -10060.364} C_VEL
LIN {X 0,Y 418.318,Z 175.378,A -85,B 0,C 180,E1 -10063.405,E2 -10063.405} C_VEL
LIN {X 0,Y 418.347,Z 175.372,A -85,B 0,C 180,E1 -10066.999,E2 -10066.999} C_VEL
LIN {X 0,Y 418.336,Z 175.373,A -85,B 0,C 180,E1 -10070.328,E2 -10070.328} C_VEL
LIN {X 0,Y 418.443,Z 175.363,A -85,B 0,C 180,E1 -10073.248,E2 -10073.248} C_VEL
LIN {X 0,Y 418.327,Z 175.379,A -85,B 0,C 180,E1 -10075.181,E2 -10075.181} C_VEL
LIN {X 0,Y 418.543,Z 175.348,A -85,B 0,C 180,E1 -10078.075,E2 -10078.075} C_VEL
LIN {X 0,Y 418.674,Z 175.332,A -85,B 0,C 180,E1 -10080,E2 -10080} C_VEL
LIN {X 0,Y 418.499,Z 175.356,A -85,B 0,C 180,E1 -10082.888,E2 -10082.888} C_VEL
LIN {X 0,Y 418.488,Z 175.354,A -85,B 0,C 180,E1 -10085.783,E2 -10085.783} C_VEL
LIN {X 0,Y 418.377,Z 175.373,A -85,B 0,C 180,E1 -10088.696,E2 -10088.696} C_VEL
LIN {X 0,Y 418.329,Z 175.374,A -85,B 0,C 180,E1 -10091.631,E2 -10091.631} C_VEL
LIN {X 0,Y 418.307,Z 175.38,A -85,B 0,C 180,E1 -10094.597,E2 -10094.597} C_VEL
LIN {X 0,Y 418.287,Z 175.38,A -85,B 0,C 180,E1 -10097.604,E2 -10097.604} C_VEL
LIN {X 0,Y 418.251,Z 175.386,A -85,B 0,C 180,E1 -10100.663,E2 -10100.663} C_VEL
LIN {X 0,Y 418.275,Z 175.382,A -85,B 0,C 180,E1 -10103.782,E2 -10103.782} C_VEL
LIN {X 0,Y 418.311,Z 175.376,A -85,B 0,C 180,E1 -10107.07,E2 -10107.07} C_VEL
LIN {X 0,Y 418.246,Z 175.388,A -85,B 0,C 180,E1 -10110.272,E2 -10110.272} C_VEL
LIN {X 0,Y 418.249,Z 175.388,A -85,B 0,C 180,E1 -10113.677,E2 -10113.677} C_VEL
LIN {X 0,Y 418.233,Z 175.388,A -85,B 0,C 180,E1 -10117.225,E2 -10117.225} C_VEL
LIN {X 0,Y 418.229,Z 175.39,A -85,B 0,C 180,E1 -10119.685,E2 -10119.685} C_VEL
LIN {X 0,Y 418.23,Z 175.386,A -85,B 0,C 180,E1 -10122.321,E2 -10122.321} C_VEL
LIN {X 0,Y 418.237,Z 175.39,A -85,B 0,C 180,E1 -10125.109,E2 -10125.109} C_VEL
LIN {X 0,Y 418.257,Z 175.387,A -85,B 0,C 180,E1 -10128.896,E2 -10128.896} C_VEL
LIN {X 0,Y 419.048,Z 179.858,A -85,B 0,C 180,E1 -10131.644,E2 -10131.644} C_VEL
LIN {X 0,Y 419.517,Z 184.307,A -85,B 0,C 180,E1 -10134.102,E2 -10134.102} C_VEL
LIN {X 0,Y 419.353,Z 188.755,A -85,B 0,C 180,E1 -10136.423,E2 -10136.423} C_VEL
LIN {X 0,Y 419.069,Z 193.457,A -85,B 0,C 180,E1 -10138.793,E2 -10138.793} C_VEL
LIN {X 0,Y 418.744,Z 198.813,A -85,B 0,C 180,E1 -10141.423,E2 -10141.423} C_VEL
LIN {X 0,Y 418.365,Z 205.544,A -85,B 0,C 180,E1 -10144.636,E2 -10144.636} C_VEL
LIN {X 0,Y 418.041,Z 211.874,A -85,B 0,C 180,E1 -10147.615,E2 -10147.615} C_VEL
LIN {X 0,Y 417.765,Z 218.893,A -85,B 0,C 180,E1 -10150.872,E2 -10150.872} C_VEL
LIN {X 0,Y 417.616,Z 222.987,A -85,B 0,C 180,E1 -10152.729,E2 -10152.729} C_VEL
LIN {X 0,Y 420.074,Z 236.468,A -85,B 0,C 180,E1 -10153.237,E2 -10153.237} C_VEL
LIN {X 0,Y 421.843,Z 248.467,A -85,B 0,C 180,E1 -10153.858,E2 -10153.858} C_VEL
LIN {X 0,Y 421.208,Z 261.322,A -85,B 0,C 180,E1 -10154.64,E2 -10154.64} C_VEL
LIN {X 0,Y 420.403,Z 273.132,A -85,B 0,C 180,E1 -10155.583,E2 -10155.583} C_VEL
LIN {X 0,Y 419.675,Z 283.992,A -85,B 0,C 180,E1 -10156.687,E2 -10156.687} C_VEL
LIN {X 0,Y 419.03,Z 293.61,A -85,B 0,C 180,E1 -10157.898,E2 -10157.898} C_VEL
LIN {X 0,Y 418.419,Z 301.494,A -85,B 0,C 180,E1 -10159.108,E2 -10159.108} C_VEL
LIN {X 0,Y 417.903,Z 309.196,A -85,B 0,C 180,E1 -10160.562,E2 -10160.562} C_VEL
LIN {X 0,Y 417.412,Z 316.296,A -85,B 0,C 180,E1 -10162.259,E2 -10162.259} C_VEL
LIN {X 0,Y 417.226,Z 320.788,A -85,B 0,C 180,E1 -10163.634,E2 -10163.634} C_VEL
LIN {X 0,Y 417.151,Z 324.637,A -85,B 0,C 180,E1 -10165.168,E2 -10165.168} C_VEL
LIN {X 0,Y 417.023,Z 326.498,A -85,B 0,C 180,E1 -10166.134,E2 -10166.134} C_VEL
LIN {X 0,Y 417.023,Z 327.897,A -85,B 0,C 180,E1 -10167.102,E2 -10167.102} C_VEL
LIN {X 0,Y 417.053,Z 328.896,A -85,B 0,C 180,E1 -10168.068,E2 -10168.068} C_VEL
LIN {X 0,Y 416.992,Z 329.503,A -85,B 0,C 180,E1 -10169.034,E2 -10169.034} C_VEL
LIN {X 0,Y 416.963,Z 329.72,A -85,B 0,C 180,E1 -10170,E2 -10170} C_VEL
LIN {X 0,Y 417.052,Z 328.898,A -85,B 0,C 180,E1 -10171.931,E2 -10171.931} C_VEL
LIN {X 0,Y 417.023,Z 327.901,A -85,B 0,C 180,E1 -10172.898,E2 -10172.898} C_VEL
LIN {X 0,Y 417.023,Z 326.503,A -85,B 0,C 180,E1 -10173.865,E2 -10173.865} C_VEL
LIN {X 0,Y 417.165,Z 323.567,A -85,B 0,C 180,E1 -10175.316,E2 -10175.316} C_VEL
LIN {X 0,Y 417.275,Z 319.589,A -85,B 0,C 180,E1 -10176.771,E2 -10176.771} C_VEL
LIN {X 0,Y 417.629,Z 313.478,A -85,B 0,C 180,E1 -10178.467,E2 -10178.467} C_VEL
LIN {X 0,Y 418.043,Z 306.799,A -85,B 0,C 180,E1 -10179.922,E2 -10179.922} C_VEL
LIN {X 0,Y 418.61,Z 298.513,A -85,B 0,C 180,E1 -10181.377,E2 -10181.377} C_VEL
LIN {X 0,Y 419.315,Z 290.026,A -85,B 0,C 180,E1 -10182.585,E2 -10182.585} C_VEL
LIN {X 0,Y 420.066,Z 279.594,A -85,B 0,C 180,E1 -10183.787,E2 -10183.787} C_VEL
LIN {X 0,Y 420.644,Z 269.159,A -85,B 0,C 180,E1 -10184.761,E2 -10184.761} C_VEL
LIN {X 0,Y 421.402,Z 257.788,A -85,B 0,C 180,E1 -10185.6,E2 -10185.6} C_VEL
LIN {X 0,Y 421.84,Z 248.465,A -85,B 0,C 180,E1 -10186.142,E2 -10186.142} C_VEL
LIN {X 0,Y 419.895,Z 235.52,A -85,B 0,C 180,E1 -10186.806,E2 -10186.806} C_VEL
LIN {X 0,Y 417.608,Z 222.861,A -85,B 0,C 180,E1 -10187.292,E2 -10187.292} C_VEL
LIN {X 0,Y 417.898,Z 215.543,A -85,B 0,C 180,E1 -10190.681,E2 -10190.681} C_VEL
LIN {X 0,Y 418.251,Z 207.776,A -85,B 0,C 180,E1 -10194.31,E2 -10194.31} C_VEL
LIN {X 0,Y 418.568,Z 201.788,A -85,B 0,C 180,E1 -10197.139,E2 -10197.139} C_VEL
LIN {X 0,Y 418.968,Z 195.439,A -85,B 0,C 180,E1 -10200.214,E2 -10200.214} C_VEL
LIN {X 0,Y 419.302,Z 189.742,A -85,B 0,C 180,E1 -10203.064,E2 -10203.064} C_VEL
LIN {X 0,Y 419.584,Z 185.395,A -85,B 0,C 180,E1 -10205.309,E2 -10205.309} C_VEL
LIN {X 0,Y 419.146,Z 180.502,A -85,B 0,C 180,E1 -10207.994,E2 -10207.994} C_VEL
LIN {X 0,Y 418.245,Z 175.391,A -85,B 0,C 180,E1 -10211.025,E2 -10211.025} C_VEL
LIN {X 0,Y 418.209,Z 175.395,A -85,B 0,C 180,E1 -10213.729,E2 -10213.729} C_VEL
LIN {X 0,Y 418.207,Z 175.392,A -85,B 0,C 180,E1 -10216.448,E2 -10216.448} C_VEL
LIN {X 0,Y 418.217,Z 175.389,A -85,B 0,C 180,E1 -10219.131,E2 -10219.131} C_VEL
LIN {X 0,Y 418.217,Z 175.391,A -85,B 0,C 180,E1 -10222.168,E2 -10222.168} C_VEL
LIN {X 0,Y 418.262,Z 175.383,A -85,B 0,C 180,E1 -10225.42,E2 -10225.42} C_VEL
LIN {X 0,Y 418.21,Z 175.392,A -85,B 0,C 180,E1 -10228.604,E2 -10228.604} C_VEL
LIN {X 0,Y 418.289,Z 175.383,A -85,B 0,C 180,E1 -10231.936,E2 -10231.936} C_VEL
LIN {X 0,Y 418.288,Z 175.379,A -85,B 0,C 180,E1 -10235.162,E2 -10235.162} C_VEL
LIN {X 0,Y 418.232,Z 175.387,A -85,B 0,C 180,E1 -10238.303,E2 -10238.303} C_VEL
LIN {X 0,Y 418.282,Z 175.384,A -85,B 0,C 180,E1 -10241.383,E2 -10241.383} C_VEL
LIN {X 0,Y 418.3,Z 175.378,A -85,B 0,C 180,E1 -10244.406,E2 -10244.406} C_VEL
LIN {X 0,Y 418.353,Z 175.375,A -85,B 0,C 180,E1 -10247.386,E2 -10247.386} C_VEL
LIN {X 0,Y 418.332,Z 175.373,A -85,B 0,C 180,E1 -10250.328,E2 -10250.328} C_VEL
LIN {X 0,Y 418.44,Z 175.364,A -85,B 0,C 180,E1 -10253.248,E2 -10253.248} C_VEL
LIN {X 0,Y 418.327,Z 175.378,A -85,B 0,C 180,E1 -10255.181,E2 -10255.181} C_VEL
LIN {X 0,Y 418.54,Z 175.348,A -85,B 0,C 180,E1 -10258.075,E2 -10258.075} C_VEL
LIN {X 0,Y 418.671,Z 175.332,A -85,B 0,C 180,E1 -10260,E2 -10260} C_VEL
LIN {X 0,Y 418.496,Z 175.358,A -85,B 0,C 180,E1 -10262.888,E2 -10262.888} C_VEL
LIN {X 0,Y 418.439,Z 175.363,A -85,B 0,C 180,E1 -10266.577,E2 -10266.577} C_VEL
LIN {X 0,Y 418.333,Z 175.373,A -85,B 0,C 180,E1 -10269.672,E2 -10269.672} C_VEL
LIN {X 0,Y 418.344,Z 175.373,A -85,B 0,C 180,E1 -10273.001,E2 -10273.001} C_VEL
LIN {X 0,Y 418.311,Z 175.378,A -85,B 0,C 180,E1 -10276.736,E2 -10276.736} C_VEL
LIN {X 0,Y 418.269,Z 175.385,A -85,B 0,C 180,E1 -10279.79,E2 -10279.79} C_VEL
LIN {X 0,Y 418.236,Z 175.385,A -85,B 0,C 180,E1 -10282.736,E2 -10282.736} C_VEL
LIN {X 0,Y 418.267,Z 175.386,A -85,B 0,C 180,E1 -10285.904,E2 -10285.904} C_VEL
LIN {X 0,Y 418.263,Z 175.384,A -85,B 0,C 180,E1 -10289.162,E2 -10289.162} C_VEL
LIN {X 0,Y 418.256,Z 175.385,A -85,B 0,C 180,E1 -10292.844,E2 -10292.844} C_VEL
LIN {X 0,Y 418.238,Z 175.386,A -85,B 0,C 180,E1 -10296.237,E2 -10296.237} C_VEL
LIN {X 0,Y 418.232,Z 175.387,A -85,B 0,C 180,E1 -10299.684,E2 -10299.684} C_VEL
LIN {X 0,Y 418.229,Z 175.386,A -85,B 0,C 180,E1 -10302.322,E2 -10302.322} C_VEL
LIN {X 0,Y 418.235,Z 175.389,A -85,B 0,C 180,E1 -10305.109,E2 -10305.109} C_VEL
LIN {X 0,Y 418.24,Z 175.386,A -85,B 0,C 180,E1 -10307.767,E2 -10307.767} C_VEL
LIN {X 0,Y 418.241,Z 175.389,A -85,B 0,C 180,E1 -10310.622,E2 -10310.622} C_VEL
LIN {X 0,Y 418.165,Z 175.399,A -85,B 0,C 180,E1 -10313.778,E2 -10313.778} C_VEL
LIN {X 0,Y 418.122,Z 177.035,A -85,B 0,C 180,E1 -10315.449,E2 -10315.449} C_VEL
LIN {X 0,Y 418.01,Z 180.971,A -85,B 0,C 180,E1 -10318.587,E2 -10318.587} C_VEL
LIN {X 0,Y 417.857,Z 185.259,A -85,B 0,C 180,E1 -10321.905,E2 -10321.905} C_VEL
LIN {X 0,Y 417.709,Z 189.776,A -85,B 0,C 180,E1 -10325.307,E2 -10325.307} C_VEL
LIN {X 0,Y 417.584,Z 193.854,A -85,B 0,C 180,E1 -10328.268,E2 -10328.268} C_VEL
LIN {X 0,Y 417.421,Z 198.254,A -85,B 0,C 180,E1 -10331.344,E2 -10331.344} C_VEL
LIN {X 0,Y 417.382,Z 200.513,A -85,B 0,C 180,E1 -10332.799,E2 -10332.799} C_VEL
LIN {X 0,Y 420.442,Z 213.605,A -85,B 0,C 180,E1 -10333.354,E2 -10333.354} C_VEL
LIN {X 0,Y 422.216,Z 224.038,A -85,B 0,C 180,E1 -10333.916,E2 -10333.916} C_VEL
LIN {X 0,Y 421.521,Z 236.258,A -85,B 0,C 180,E1 -10334.652,E2 -10334.652} C_VEL
LIN {X 0,Y 420.9,Z 247.021,A -85,B 0,C 180,E1 -10335.495,E2 -10335.495} C_VEL
LIN {X 0,Y 420.258,Z 257.986,A -85,B 0,C 180,E1 -10336.584,E2 -10336.584} C_VEL
LIN {X 0,Y 419.588,Z 266.889,A -85,B 0,C 180,E1 -10337.669,E2 -10337.669} C_VEL
LIN {X 0,Y 418.984,Z 275.054,A -85,B 0,C 180,E1 -10338.878,E2 -10338.878} C_VEL
LIN {X 0,Y 418.376,Z 283.053,A -85,B 0,C 180,E1 -10340.33,E2 -10340.33} C_VEL
LIN {X 0,Y 417.848,Z 289.475,A -85,B 0,C 180,E1 -10341.781,E2 -10341.781} C_VEL
LIN {X 0,Y 417.543,Z 295.548,A -85,B 0,C 180,E1 -10343.57,E2 -10343.57} C_VEL
LIN {X 0,Y 417.234,Z 299.583,A -85,B 0,C 180,E1 -10345.169,E2 -10345.169} C_VEL
LIN {X 0,Y 417.176,Z 301.442,A -85,B 0,C 180,E1 -10346.136,E2 -10346.136} C_VEL
LIN {X 0,Y 417.185,Z 302.84,A -85,B 0,C 180,E1 -10347.103,E2 -10347.103} C_VEL
LIN {X 0,Y 417.015,Z 304.453,A -85,B 0,C 180,E1 -10349.035,E2 -10349.035} C_VEL
LIN {X 0,Y 417.006,Z 304.687,A -85,B 0,C 180,E1 -10350,E2 -10350} C_VEL
LIN {X 0,Y 417.015,Z 304.499,A -85,B 0,C 180,E1 -10350.966,E2 -10350.966} C_VEL
LIN {X 0,Y 417.185,Z 302.946,A -85,B 0,C 180,E1 -10352.897,E2 -10352.897} C_VEL
LIN {X 0,Y 417.172,Z 301.594,A -85,B 0,C 180,E1 -10353.864,E2 -10353.864} C_VEL
LIN {X 0,Y 417.278,Z 299.237,A -85,B 0,C 180,E1 -10355.083,E2 -10355.083} C_VEL
LIN {X 0,Y 416.759,Z 297.46,A -85,B 0,C 180,E1 -10355.852,E2 -10355.852} C_VEL
LIN {X 0,Y 414.087,Z 294.136,A -85,B 0,C 180,E1 -10357.087,E2 -10357.087} C_VEL
LIN {X 0,Y 411.45,Z 290.202,A -85,B 0,C 180,E1 -10358.301,E2 -10358.301} C_VEL
LIN {X 0,Y 411,Z 287.371,A -85,B 0,C 180,E1 -10359.027,E2 -10359.027} C_VEL
LIN {X 0,Y 411.598,Z 280.005,A -85,B 0,C 180,E1 -10360.577,E2 -10360.577} C_VEL
LIN {X 0,Y 412.323,Z 271.195,A -85,B 0,C 180,E1 -10362.052,E2 -10362.052} C_VEL
LIN {X 0,Y 413.093,Z 262.153,A -85,B 0,C 180,E1 -10363.278,E2 -10363.278} C_VEL
LIN {X 0,Y 413.75,Z 252.108,A -85,B 0,C 180,E1 -10364.388,E2 -10364.388} C_VEL
LIN {X 0,Y 414.427,Z 241.008,A -85,B 0,C 180,E1 -10365.366,E2 -10365.366} C_VEL
LIN {X 0,Y 415.193,Z 229.008,A -85,B 0,C 180,E1 -10366.186,E2 -10366.186} C_VEL
LIN {X 0,Y 415.31,Z 223.89,A -85,B 0,C 180,E1 -10366.477,E2 -10366.477} C_VEL
LIN {X 0,Y 412.918,Z 211.566,A -85,B 0,C 180,E1 -10367.15,E2 -10367.15} C_VEL
LIN {X 0,Y 410.3,Z 200.569,A -85,B 0,C 180,E1 -10367.624,E2 -10367.624} C_VEL
LIN {X 0,Y 410.392,Z 197.101,A -85,B 0,C 180,E1 -10370.03,E2 -10370.03} C_VEL
LIN {X 0,Y 410.555,Z 192.753,A -85,B 0,C 180,E1 -10373.186,E2 -10373.186} C_VEL
LIN {X 0,Y 410.695,Z 188.422,A -85,B 0,C 180,E1 -10376.419,E2 -10376.419} C_VEL
LIN {X 0,Y 410.89,Z 184.153,A -85,B 0,C 180,E1 -10379.738,E2 -10379.738} C_VEL
LIN {X 0,Y 411.069,Z 179.821,A -85,B 0,C 180,E1 -10383.168,E2 -10383.168} C_VEL
LIN {X 0,Y 411.101,Z 176.92,A -85,B 0,C 180,E1 -10385.539,E2 -10385.539} C_VEL
LIN {X 0,Y 411.161,Z 176.272,A -85,B 0,C 180,E1 -10386.745,E2 -10386.745} C_VEL
LIN {X 0,Y 411.169,Z 176.269,A -85,B 0,C 180,E1 -10389.72,E2 -10389.72} C_VEL
LIN {X 0,Y 411.166,Z 176.27,A -85,B 0,C 180,E1 -10393.135,E2 -10393.135} C_VEL
LIN {X 0,Y 411.169,Z 176.266,A -85,B 0,C 180,E1 -10395.881,E2 -10395.881} C_VEL
LIN {X 0,Y 411.163,Z 176.27,A -85,B 0,C 180,E1 -10398.772,E2 -10398.772} C_VEL
LIN {X 0,Y 411.186,Z 176.264,A -85,B 0,C 180,E1 -10402.025,E2 -10402.025} C_VEL
LIN {X 0,Y 411.193,Z 176.263,A -85,B 0,C 180,E1 -10405.665,E2 -10405.665} C_VEL
LIN {X 0,Y 411.191,Z 176.264,A -85,B 0,C 180,E1 -10409.152,E2 -10409.152} C_VEL
LIN {X 0,Y 411.26,Z 176.259,A -85,B 0,C 180,E1 -10412.522,E2 -10412.522} C_VEL
LIN {X 0,Y 411.227,Z 176.26,A -85,B 0,C 180,E1 -10415.784,E2 -10415.784} C_VEL
LIN {X 0,Y 411.198,Z 176.262,A -85,B 0,C 180,E1 -10418.966,E2 -10418.966} C_VEL
LIN {X 0,Y 411.252,Z 176.259,A -85,B 0,C 180,E1 -10422.085,E2 -10422.085} C_VEL
LIN {X 0,Y 411.261,Z 176.255,A -85,B 0,C 180,E1 -10425.147,E2 -10425.147} C_VEL
LIN {X 0,Y 411.283,Z 176.253,A -85,B 0,C 180,E1 -10428.167,E2 -10428.167} C_VEL
LIN {X 0,Y 411.317,Z 176.249,A -85,B 0,C 180,E1 -10431.154,E2 -10431.154} C_VEL
LIN {X 0,Y 411.432,Z 176.234,A -85,B 0,C 180,E1 -10434.117,E2 -10434.117} C_VEL
LIN {X 0,Y 411.511,Z 176.224,A -85,B 0,C 180,E1 -10438.043,E2 -10438.043} C_VEL
LIN {X 0,Y 411.643,Z 176.207,A -85,B 0,C 180,E1 -10440,E2 -10440} C_VEL
LIN {X 0,Y 411.456,Z 176.234,A -85,B 0,C 180,E1 -10442.937,E2 -10442.937} C_VEL
LIN {X 0,Y 411.433,Z 176.232,A -85,B 0,C 180,E1 -10445.883,E2 -10445.883} C_VEL
LIN {X 0,Y 411.318,Z 176.252,A -85,B 0,C 180,E1 -10448.846,E2 -10448.846} C_VEL
LIN {X 0,Y 411.297,Z 176.25,A -85,B 0,C 180,E1 -10451.832,E2 -10451.832} C_VEL
LIN {X 0,Y 411.263,Z 176.258,A -85,B 0,C 180,E1 -10454.853,E2 -10454.853} C_VEL
LIN {X 0,Y 411.252,Z 176.258,A -85,B 0,C 180,E1 -10457.915,E2 -10457.915} C_VEL
LIN {X 0,Y 411.197,Z 176.262,A -85,B 0,C 180,E1 -10461.034,E2 -10461.034} C_VEL
LIN {X 0,Y 411.221,Z 176.264,A -85,B 0,C 180,E1 -10464.216,E2 -10464.216} C_VEL
LIN {X 0,Y 411.26,Z 176.256,A -85,B 0,C 180,E1 -10467.478,E2 -10467.478} C_VEL
LIN {X 0,Y 411.19,Z 176.264,A -85,B 0,C 180,E1 -10470.848,E2 -10470.848} C_VEL
LIN {X 0,Y 411.206,Z 176.262,A -85,B 0,C 180,E1 -10474.334,E2 -10474.334} C_VEL
LIN {X 0,Y 411.182,Z 176.266,A -85,B 0,C 180,E1 -10477.975,E2 -10477.975} C_VEL
LIN {X 0,Y 411.163,Z 176.271,A -85,B 0,C 180,E1 -10481.228,E2 -10481.228} C_VEL
LIN {X 0,Y 411.177,Z 176.269,A -85,B 0,C 180,E1 -10484.49,E2 -10484.49} C_VEL
LIN {X 0,Y 411.201,Z 176.264,A -85,B 0,C 180,E1 -10488.197,E2 -10488.197} C_VEL
LIN {X 0,Y 411.215,Z 176.3,A -85,B 0,C 180,E1 -10488.764,E2 -10488.764} C_VEL
LIN {X 0,Y 412.084,Z 181.165,A -85,B 0,C 180,E1 -10491.677,E2 -10491.677} C_VEL
LIN {X 0,Y 412.508,Z 185.305,A -85,B 0,C 180,E1 -10494,E2 -10494} C_VEL
LIN {X 0,Y 412.456,Z 188.633,A -85,B 0,C 180,E1 -10495.785,E2 -10495.785} C_VEL
